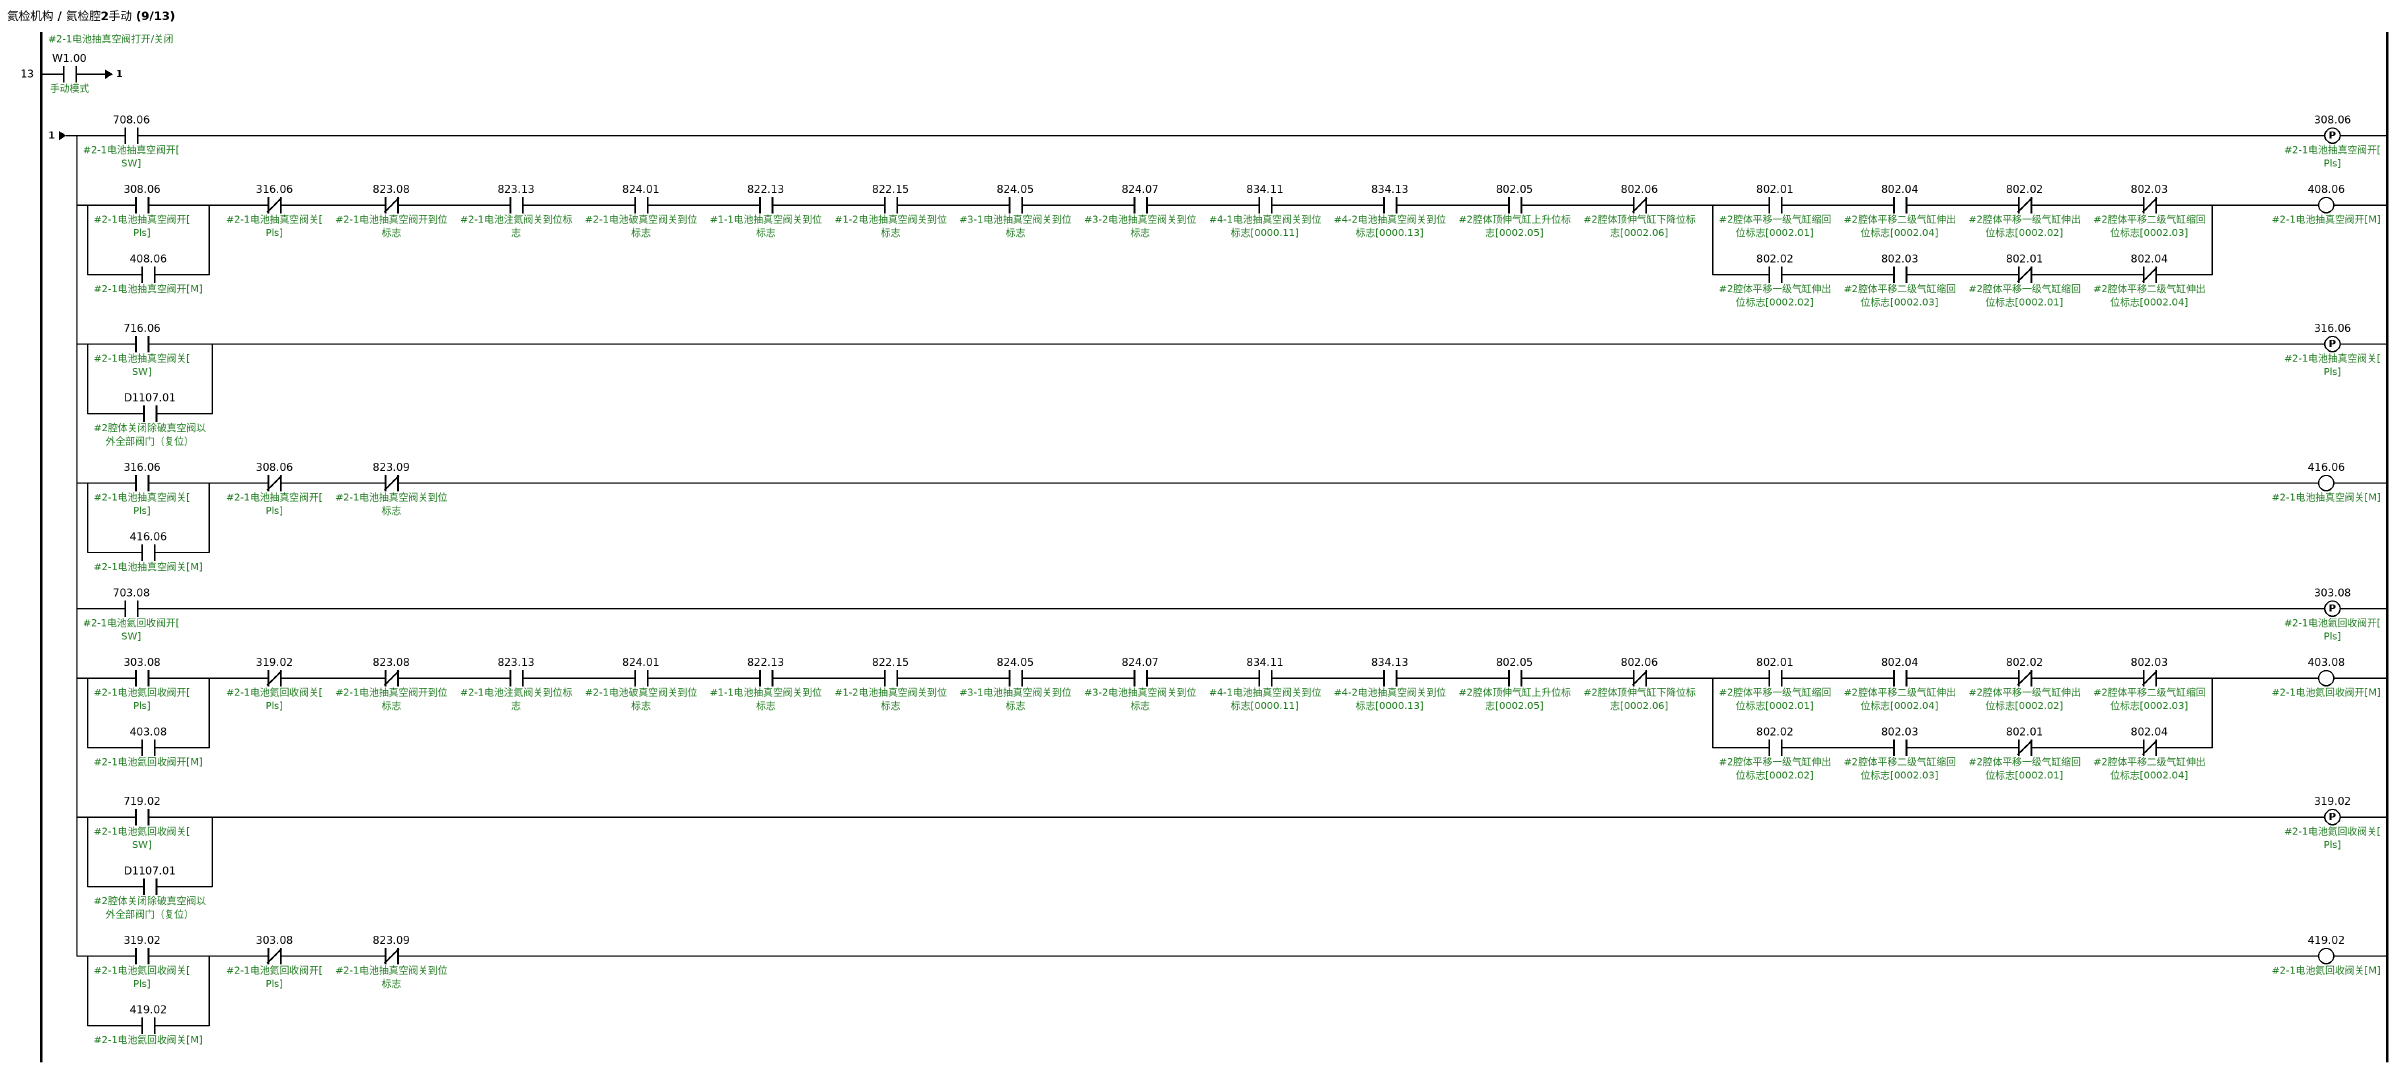
; [picture p192: 氦检机构 / 氦检腔2手动, rungs 13-13]
; rung 13: #2-1电池抽真空阀打开/关闭
LD W1.00  ; 手动模式
OUT TR0
AND 708.06  ; #2-1电池抽真空阀开[SW]
DIFU(013) 308.06  ; #2-1电池抽真空阀开[Pls]
LD TR0
LD 308.06  ; #2-1电池抽真空阀开[Pls]
OR 408.06  ; #2-1电池抽真空阀开[M]
ANDLD
ANDNOT 316.06  ; #2-1电池抽真空阀关[Pls]
ANDNOT 823.08  ; #2-1电池抽真空阀开到位标志
AND 823.13  ; #2-1电池注氦阀关到位标志
AND 824.01  ; #2-1电池破真空阀关到位标志
AND 822.13  ; #1-1电池抽真空阀关到位标志
AND 822.15  ; #1-2电池抽真空阀关到位标志
AND 824.05  ; #3-1电池抽真空阀关到位标志
AND 824.07  ; #3-2电池抽真空阀关到位标志
AND 834.11  ; #4-1电池抽真空阀关到位标志[0000.11]
AND 834.13  ; #4-2电池抽真空阀关到位标志[0000.13]
AND 802.05  ; #2腔体顶伸气缸上升位标志[0002.05]
ANDNOT 802.06  ; #2腔体顶伸气缸下降位标志[0002.06]
LD 802.01  ; #2腔体平移一级气缸缩回位标志[0002.01]
AND 802.04  ; #2腔体平移二级气缸伸出位标志[0002.04]
ANDNOT 802.02  ; #2腔体平移一级气缸伸出位标志[0002.02]
ANDNOT 802.03  ; #2腔体平移二级气缸缩回位标志[0002.03]
LD 802.02  ; #2腔体平移一级气缸伸出位标志[0002.02]
AND 802.03  ; #2腔体平移二级气缸缩回位标志[0002.03]
ANDNOT 802.01  ; #2腔体平移一级气缸缩回位标志[0002.01]
ANDNOT 802.04  ; #2腔体平移二级气缸伸出位标志[0002.04]
ORLD
ANDLD
OUT 408.06  ; #2-1电池抽真空阀开[M]
LD TR0
LD 716.06  ; #2-1电池抽真空阀关[SW]
OR D1107.01  ; #2腔体关闭除破真空阀以外全部阀门（复位）
ANDLD
DIFU(013) 316.06  ; #2-1电池抽真空阀关[Pls]
LD TR0
LD 316.06  ; #2-1电池抽真空阀关[Pls]
OR 416.06  ; #2-1电池抽真空阀关[M]
ANDLD
ANDNOT 308.06  ; #2-1电池抽真空阀开[Pls]
ANDNOT 823.09  ; #2-1电池抽真空阀关到位标志
OUT 416.06  ; #2-1电池抽真空阀关[M]
LD TR0
AND 703.08  ; #2-1电池氦回收阀开[SW]
DIFU(013) 303.08  ; #2-1电池氦回收阀开[Pls]
LD TR0
LD 303.08  ; #2-1电池氦回收阀开[Pls]
OR 403.08  ; #2-1电池氦回收阀开[M]
ANDLD
ANDNOT 319.02  ; #2-1电池氦回收阀关[Pls]
ANDNOT 823.08  ; #2-1电池抽真空阀开到位标志
AND 823.13  ; #2-1电池注氦阀关到位标志
AND 824.01  ; #2-1电池破真空阀关到位标志
AND 822.13  ; #1-1电池抽真空阀关到位标志
AND 822.15  ; #1-2电池抽真空阀关到位标志
AND 824.05  ; #3-1电池抽真空阀关到位标志
AND 824.07  ; #3-2电池抽真空阀关到位标志
AND 834.11  ; #4-1电池抽真空阀关到位标志[0000.11]
AND 834.13  ; #4-2电池抽真空阀关到位标志[0000.13]
AND 802.05  ; #2腔体顶伸气缸上升位标志[0002.05]
ANDNOT 802.06  ; #2腔体顶伸气缸下降位标志[0002.06]
LD 802.01  ; #2腔体平移一级气缸缩回位标志[0002.01]
AND 802.04  ; #2腔体平移二级气缸伸出位标志[0002.04]
ANDNOT 802.02  ; #2腔体平移一级气缸伸出位标志[0002.02]
ANDNOT 802.03  ; #2腔体平移二级气缸缩回位标志[0002.03]
LD 802.02  ; #2腔体平移一级气缸伸出位标志[0002.02]
AND 802.03  ; #2腔体平移二级气缸缩回位标志[0002.03]
ANDNOT 802.01  ; #2腔体平移一级气缸缩回位标志[0002.01]
ANDNOT 802.04  ; #2腔体平移二级气缸伸出位标志[0002.04]
ORLD
ANDLD
OUT 403.08  ; #2-1电池氦回收阀开[M]
LD TR0
LD 719.02  ; #2-1电池氦回收阀关[SW]
OR D1107.01  ; #2腔体关闭除破真空阀以外全部阀门（复位）
ANDLD
DIFU(013) 319.02  ; #2-1电池氦回收阀关[Pls]
LD TR0
LD 319.02  ; #2-1电池氦回收阀关[Pls]
OR 419.02  ; #2-1电池氦回收阀关[M]
ANDLD
ANDNOT 303.08  ; #2-1电池氦回收阀开[Pls]
ANDNOT 823.09  ; #2-1电池抽真空阀关到位标志
OUT 419.02  ; #2-1电池氦回收阀关[M]

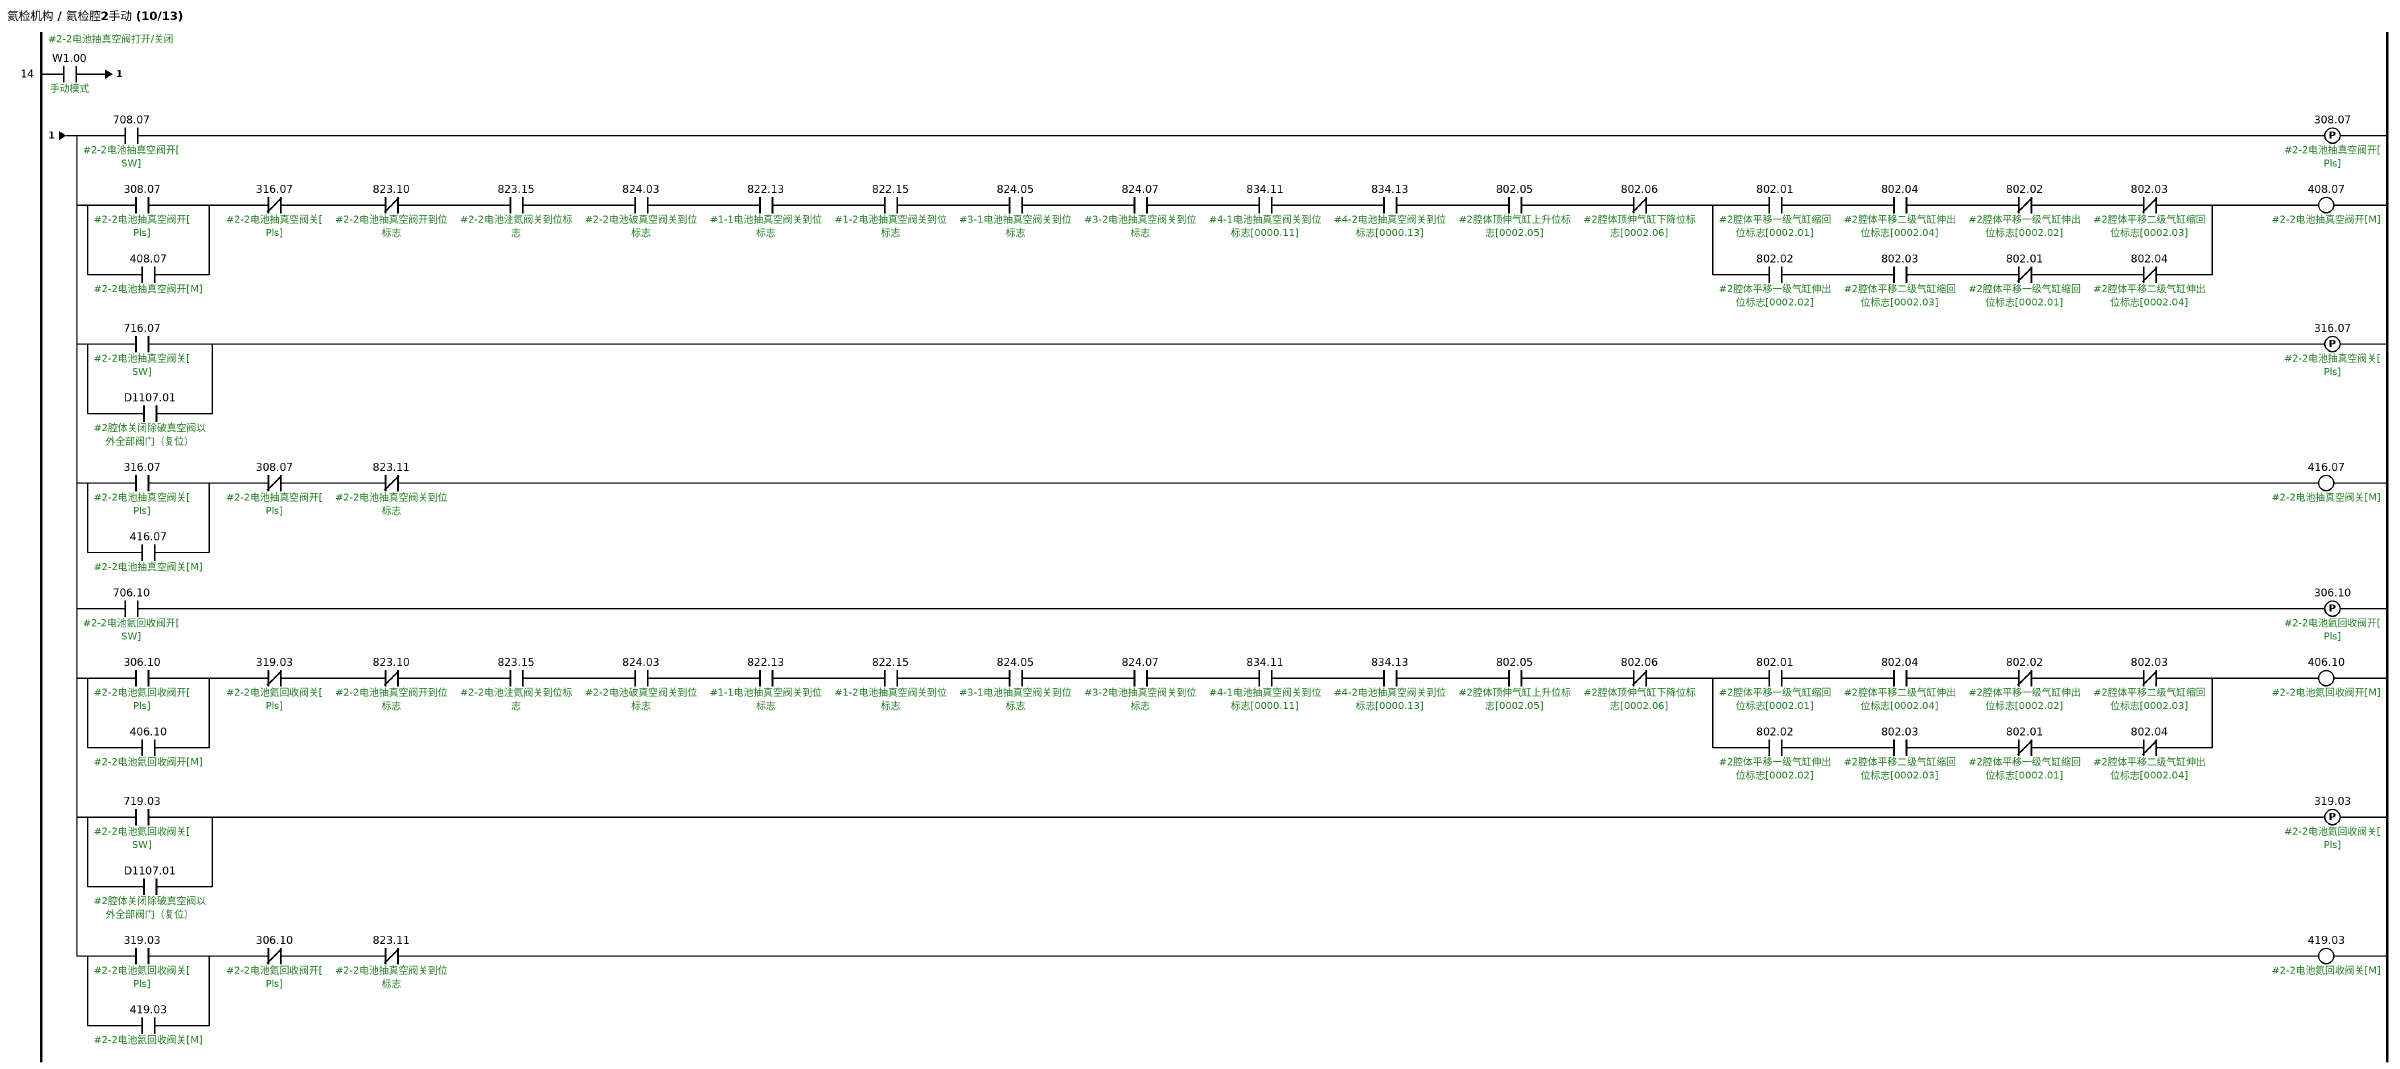
; rung 14: #2-2电池抽真空阀打开/关闭
LD W1.00  ; 手动模式
OUT TR0
AND 708.07  ; #2-2电池抽真空阀开[SW]
DIFU(013) 308.07  ; #2-2电池抽真空阀开[Pls]
LD TR0
LD 308.07  ; #2-2电池抽真空阀开[Pls]
OR 408.07  ; #2-2电池抽真空阀开[M]
ANDLD
ANDNOT 316.07  ; #2-2电池抽真空阀关[Pls]
ANDNOT 823.10  ; #2-2电池抽真空阀开到位标志
AND 823.15  ; #2-2电池注氦阀关到位标志
AND 824.03  ; #2-2电池破真空阀关到位标志
AND 822.13  ; #1-1电池抽真空阀关到位标志
AND 822.15  ; #1-2电池抽真空阀关到位标志
AND 824.05  ; #3-1电池抽真空阀关到位标志
AND 824.07  ; #3-2电池抽真空阀关到位标志
AND 834.11  ; #4-1电池抽真空阀关到位标志[0000.11]
AND 834.13  ; #4-2电池抽真空阀关到位标志[0000.13]
AND 802.05  ; #2腔体顶伸气缸上升位标志[0002.05]
ANDNOT 802.06  ; #2腔体顶伸气缸下降位标志[0002.06]
LD 802.01  ; #2腔体平移一级气缸缩回位标志[0002.01]
AND 802.04  ; #2腔体平移二级气缸伸出位标志[0002.04]
ANDNOT 802.02  ; #2腔体平移一级气缸伸出位标志[0002.02]
ANDNOT 802.03  ; #2腔体平移二级气缸缩回位标志[0002.03]
LD 802.02  ; #2腔体平移一级气缸伸出位标志[0002.02]
AND 802.03  ; #2腔体平移二级气缸缩回位标志[0002.03]
ANDNOT 802.01  ; #2腔体平移一级气缸缩回位标志[0002.01]
ANDNOT 802.04  ; #2腔体平移二级气缸伸出位标志[0002.04]
ORLD
ANDLD
OUT 408.07  ; #2-2电池抽真空阀开[M]
LD TR0
LD 716.07  ; #2-2电池抽真空阀关[SW]
OR D1107.01  ; #2腔体关闭除破真空阀以外全部阀门（复位）
ANDLD
DIFU(013) 316.07  ; #2-2电池抽真空阀关[Pls]
LD TR0
LD 316.07  ; #2-2电池抽真空阀关[Pls]
OR 416.07  ; #2-2电池抽真空阀关[M]
ANDLD
ANDNOT 308.07  ; #2-2电池抽真空阀开[Pls]
ANDNOT 823.11  ; #2-2电池抽真空阀关到位标志
OUT 416.07  ; #2-2电池抽真空阀关[M]
LD TR0
AND 706.10  ; #2-2电池氦回收阀开[SW]
DIFU(013) 306.10  ; #2-2电池氦回收阀开[Pls]
LD TR0
LD 306.10  ; #2-2电池氦回收阀开[Pls]
OR 406.10  ; #2-2电池氦回收阀开[M]
ANDLD
ANDNOT 319.03  ; #2-2电池氦回收阀关[Pls]
ANDNOT 823.10  ; #2-2电池抽真空阀开到位标志
AND 823.15  ; #2-2电池注氦阀关到位标志
AND 824.03  ; #2-2电池破真空阀关到位标志
AND 822.13  ; #1-1电池抽真空阀关到位标志
AND 822.15  ; #1-2电池抽真空阀关到位标志
AND 824.05  ; #3-1电池抽真空阀关到位标志
AND 824.07  ; #3-2电池抽真空阀关到位标志
AND 834.11  ; #4-1电池抽真空阀关到位标志[0000.11]
AND 834.13  ; #4-2电池抽真空阀关到位标志[0000.13]
AND 802.05  ; #2腔体顶伸气缸上升位标志[0002.05]
ANDNOT 802.06  ; #2腔体顶伸气缸下降位标志[0002.06]
LD 802.01  ; #2腔体平移一级气缸缩回位标志[0002.01]
AND 802.04  ; #2腔体平移二级气缸伸出位标志[0002.04]
ANDNOT 802.02  ; #2腔体平移一级气缸伸出位标志[0002.02]
ANDNOT 802.03  ; #2腔体平移二级气缸缩回位标志[0002.03]
LD 802.02  ; #2腔体平移一级气缸伸出位标志[0002.02]
AND 802.03  ; #2腔体平移二级气缸缩回位标志[0002.03]
ANDNOT 802.01  ; #2腔体平移一级气缸缩回位标志[0002.01]
ANDNOT 802.04  ; #2腔体平移二级气缸伸出位标志[0002.04]
ORLD
ANDLD
OUT 406.10  ; #2-2电池氦回收阀开[M]
LD TR0
LD 719.03  ; #2-2电池氦回收阀关[SW]
OR D1107.01  ; #2腔体关闭除破真空阀以外全部阀门（复位）
ANDLD
DIFU(013) 319.03  ; #2-2电池氦回收阀关[Pls]
LD TR0
LD 319.03  ; #2-2电池氦回收阀关[Pls]
OR 419.03  ; #2-2电池氦回收阀关[M]
ANDLD
ANDNOT 306.10  ; #2-2电池氦回收阀开[Pls]
ANDNOT 823.11  ; #2-2电池抽真空阀关到位标志
OUT 419.03  ; #2-2电池氦回收阀关[M]

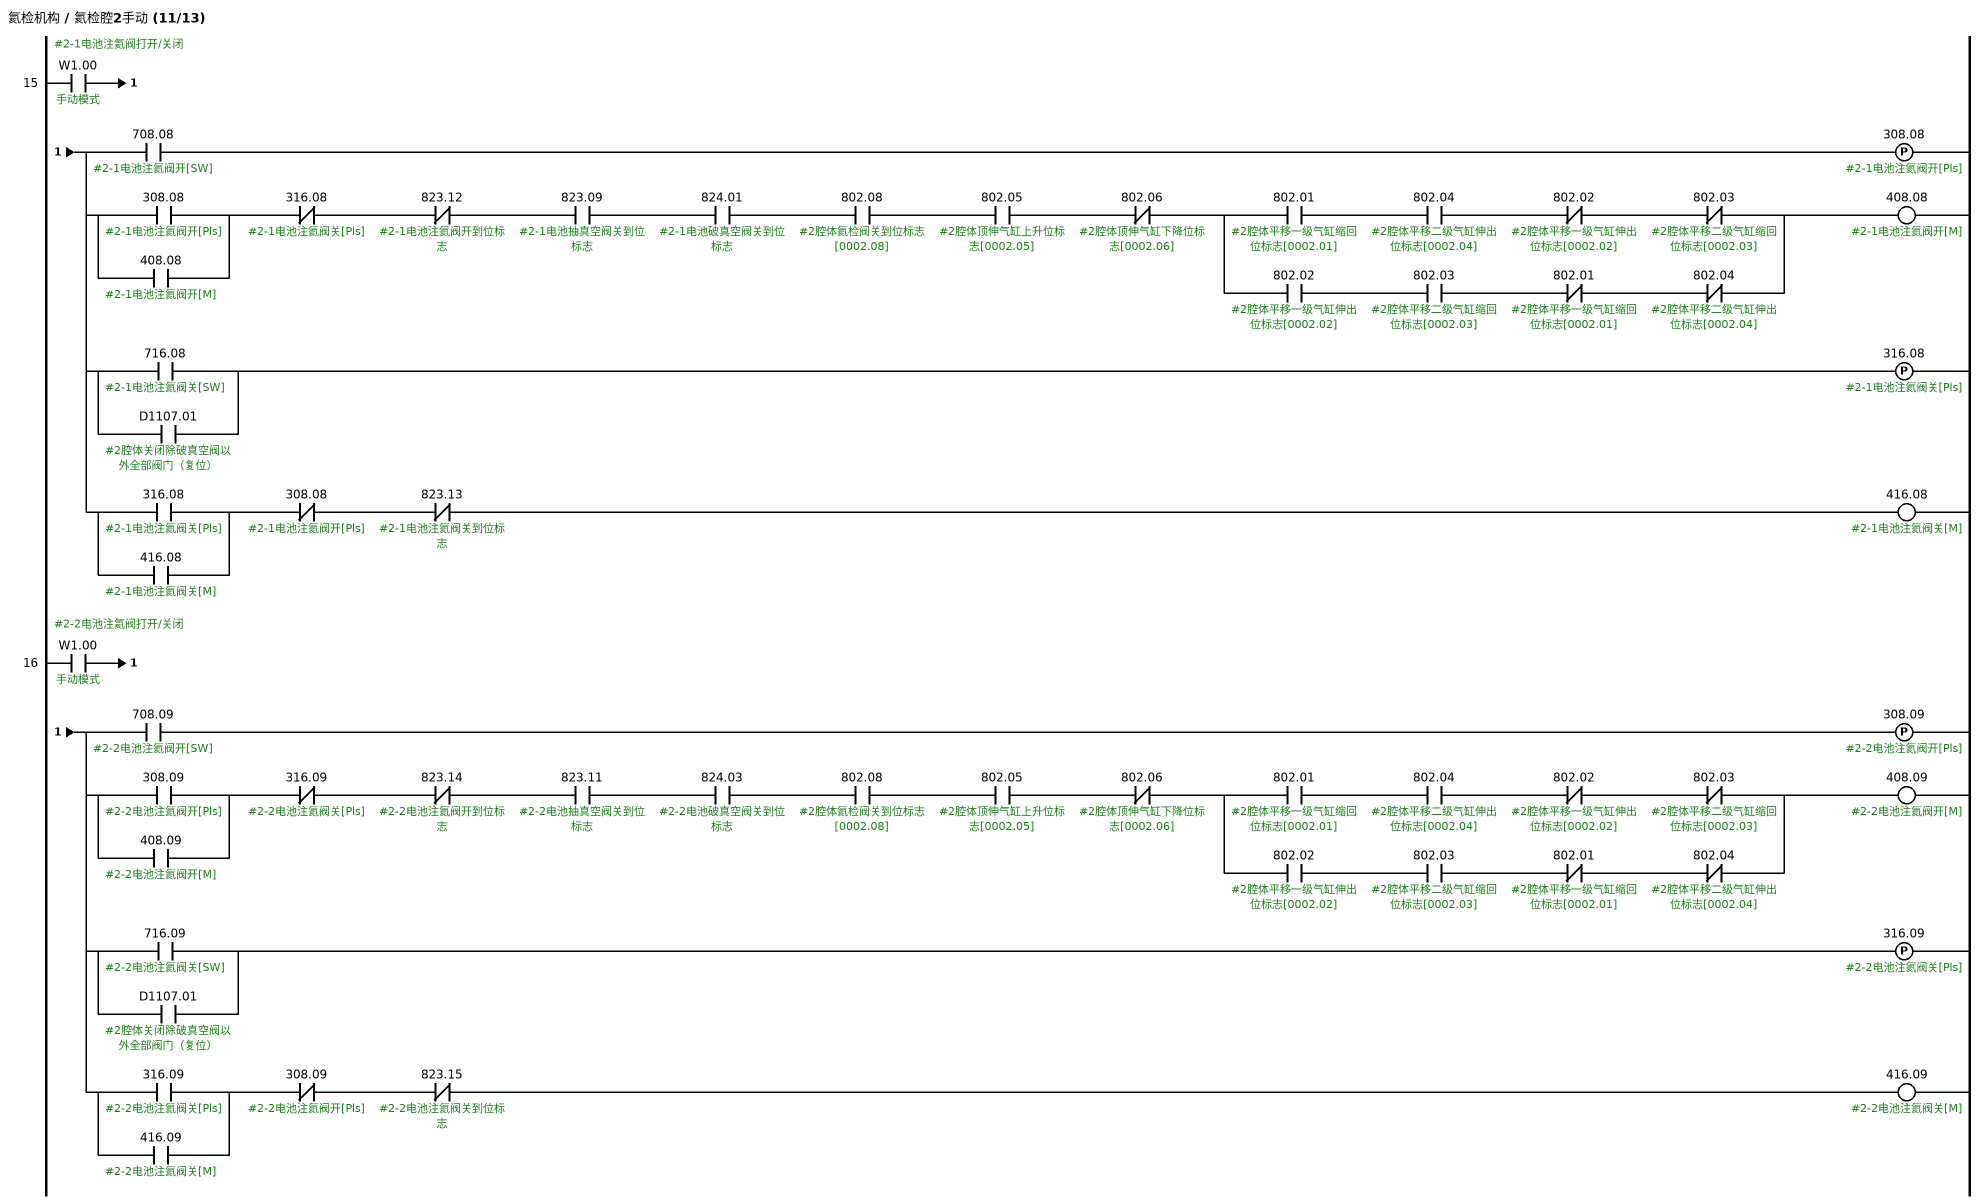
; rung 15: #2-1电池注氦阀打开/关闭
LD W1.00  ; 手动模式
OUT TR0
AND 708.08  ; #2-1电池注氦阀开[SW]
DIFU(013) 308.08  ; #2-1电池注氦阀开[Pls]
LD TR0
LD 308.08  ; #2-1电池注氦阀开[Pls]
OR 408.08  ; #2-1电池注氦阀开[M]
ANDLD
ANDNOT 316.08  ; #2-1电池注氦阀关[Pls]
ANDNOT 823.12  ; #2-1电池注氦阀开到位标志
AND 823.09  ; #2-1电池抽真空阀关到位标志
AND 824.01  ; #2-1电池破真空阀关到位标志
AND 802.08  ; #2腔体氦检阀关到位标志[0002.08]
AND 802.05  ; #2腔体顶伸气缸上升位标志[0002.05]
ANDNOT 802.06  ; #2腔体顶伸气缸下降位标志[0002.06]
LD 802.01  ; #2腔体平移一级气缸缩回位标志[0002.01]
AND 802.04  ; #2腔体平移二级气缸伸出位标志[0002.04]
ANDNOT 802.02  ; #2腔体平移一级气缸伸出位标志[0002.02]
ANDNOT 802.03  ; #2腔体平移二级气缸缩回位标志[0002.03]
LD 802.02  ; #2腔体平移一级气缸伸出位标志[0002.02]
AND 802.03  ; #2腔体平移二级气缸缩回位标志[0002.03]
ANDNOT 802.01  ; #2腔体平移一级气缸缩回位标志[0002.01]
ANDNOT 802.04  ; #2腔体平移二级气缸伸出位标志[0002.04]
ORLD
ANDLD
OUT 408.08  ; #2-1电池注氦阀开[M]
LD TR0
LD 716.08  ; #2-1电池注氦阀关[SW]
OR D1107.01  ; #2腔体关闭除破真空阀以外全部阀门（复位）
ANDLD
DIFU(013) 316.08  ; #2-1电池注氦阀关[Pls]
LD TR0
LD 316.08  ; #2-1电池注氦阀关[Pls]
OR 416.08  ; #2-1电池注氦阀关[M]
ANDLD
ANDNOT 308.08  ; #2-1电池注氦阀开[Pls]
ANDNOT 823.13  ; #2-1电池注氦阀关到位标志
OUT 416.08  ; #2-1电池注氦阀关[M]
; rung 16: #2-2电池注氦阀打开/关闭
LD W1.00  ; 手动模式
OUT TR0
AND 708.09  ; #2-2电池注氦阀开[SW]
DIFU(013) 308.09  ; #2-2电池注氦阀开[Pls]
LD TR0
LD 308.09  ; #2-2电池注氦阀开[Pls]
OR 408.09  ; #2-2电池注氦阀开[M]
ANDLD
ANDNOT 316.09  ; #2-2电池注氦阀关[Pls]
ANDNOT 823.14  ; #2-2电池注氦阀开到位标志
AND 823.11  ; #2-2电池抽真空阀关到位标志
AND 824.03  ; #2-2电池破真空阀关到位标志
AND 802.08  ; #2腔体氦检阀关到位标志[0002.08]
AND 802.05  ; #2腔体顶伸气缸上升位标志[0002.05]
ANDNOT 802.06  ; #2腔体顶伸气缸下降位标志[0002.06]
LD 802.01  ; #2腔体平移一级气缸缩回位标志[0002.01]
AND 802.04  ; #2腔体平移二级气缸伸出位标志[0002.04]
ANDNOT 802.02  ; #2腔体平移一级气缸伸出位标志[0002.02]
ANDNOT 802.03  ; #2腔体平移二级气缸缩回位标志[0002.03]
LD 802.02  ; #2腔体平移一级气缸伸出位标志[0002.02]
AND 802.03  ; #2腔体平移二级气缸缩回位标志[0002.03]
ANDNOT 802.01  ; #2腔体平移一级气缸缩回位标志[0002.01]
ANDNOT 802.04  ; #2腔体平移二级气缸伸出位标志[0002.04]
ORLD
ANDLD
OUT 408.09  ; #2-2电池注氦阀开[M]
LD TR0
LD 716.09  ; #2-2电池注氦阀关[SW]
OR D1107.01  ; #2腔体关闭除破真空阀以外全部阀门（复位）
ANDLD
DIFU(013) 316.09  ; #2-2电池注氦阀关[Pls]
LD TR0
LD 316.09  ; #2-2电池注氦阀关[Pls]
OR 416.09  ; #2-2电池注氦阀关[M]
ANDLD
ANDNOT 308.09  ; #2-2电池注氦阀开[Pls]
ANDNOT 823.15  ; #2-2电池注氦阀关到位标志
OUT 416.09  ; #2-2电池注氦阀关[M]

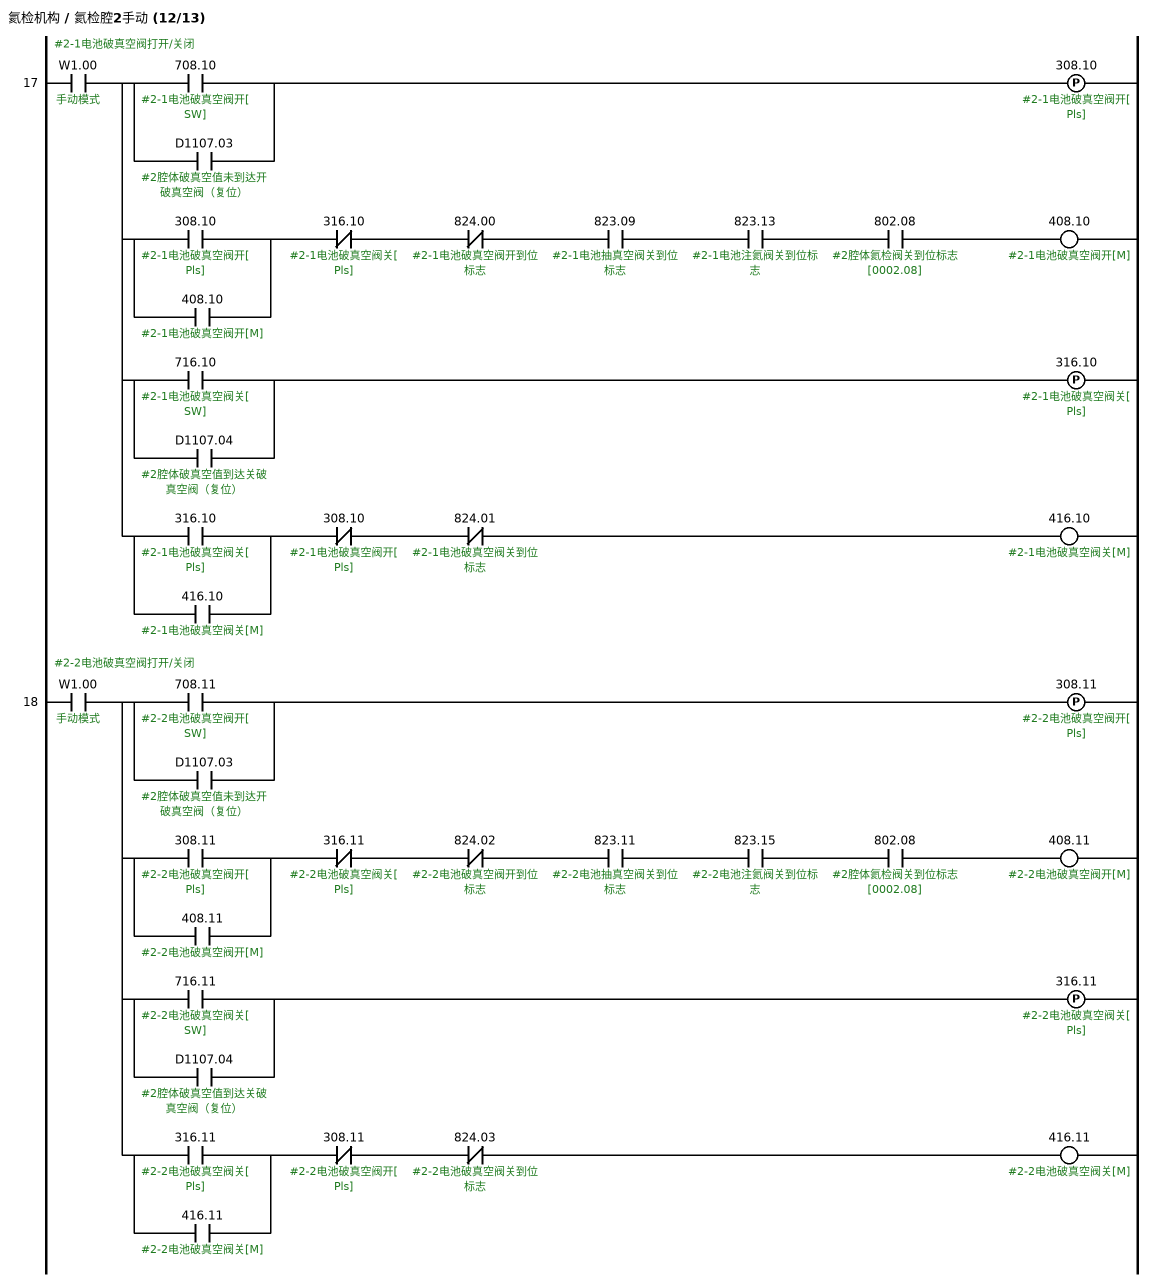
; rung 17: #2-1电池破真空阀打开/关闭
LD W1.00  ; 手动模式
OUT TR0
LD 708.10  ; #2-1电池破真空阀开[SW]
OR D1107.03  ; #2腔体破真空值未到达开破真空阀（复位）
ANDLD
DIFU(013) 308.10  ; #2-1电池破真空阀开[Pls]
LD TR0
LD 308.10  ; #2-1电池破真空阀开[Pls]
OR 408.10  ; #2-1电池破真空阀开[M]
ANDLD
ANDNOT 316.10  ; #2-1电池破真空阀关[Pls]
ANDNOT 824.00  ; #2-1电池破真空阀开到位标志
AND 823.09  ; #2-1电池抽真空阀关到位标志
AND 823.13  ; #2-1电池注氦阀关到位标志
AND 802.08  ; #2腔体氦检阀关到位标志[0002.08]
OUT 408.10  ; #2-1电池破真空阀开[M]
LD TR0
LD 716.10  ; #2-1电池破真空阀关[SW]
OR D1107.04  ; #2腔体破真空值到达关破真空阀（复位）
ANDLD
DIFU(013) 316.10  ; #2-1电池破真空阀关[Pls]
LD TR0
LD 316.10  ; #2-1电池破真空阀关[Pls]
OR 416.10  ; #2-1电池破真空阀关[M]
ANDLD
ANDNOT 308.10  ; #2-1电池破真空阀开[Pls]
ANDNOT 824.01  ; #2-1电池破真空阀关到位标志
OUT 416.10  ; #2-1电池破真空阀关[M]
; rung 18: #2-2电池破真空阀打开/关闭
LD W1.00  ; 手动模式
OUT TR0
LD 708.11  ; #2-2电池破真空阀开[SW]
OR D1107.03  ; #2腔体破真空值未到达开破真空阀（复位）
ANDLD
DIFU(013) 308.11  ; #2-2电池破真空阀开[Pls]
LD TR0
LD 308.11  ; #2-2电池破真空阀开[Pls]
OR 408.11  ; #2-2电池破真空阀开[M]
ANDLD
ANDNOT 316.11  ; #2-2电池破真空阀关[Pls]
ANDNOT 824.02  ; #2-2电池破真空阀开到位标志
AND 823.11  ; #2-2电池抽真空阀关到位标志
AND 823.15  ; #2-2电池注氦阀关到位标志
AND 802.08  ; #2腔体氦检阀关到位标志[0002.08]
OUT 408.11  ; #2-2电池破真空阀开[M]
LD TR0
LD 716.11  ; #2-2电池破真空阀关[SW]
OR D1107.04  ; #2腔体破真空值到达关破真空阀（复位）
ANDLD
DIFU(013) 316.11  ; #2-2电池破真空阀关[Pls]
LD TR0
LD 316.11  ; #2-2电池破真空阀关[Pls]
OR 416.11  ; #2-2电池破真空阀关[M]
ANDLD
ANDNOT 308.11  ; #2-2电池破真空阀开[Pls]
ANDNOT 824.03  ; #2-2电池破真空阀关到位标志
OUT 416.11  ; #2-2电池破真空阀关[M]

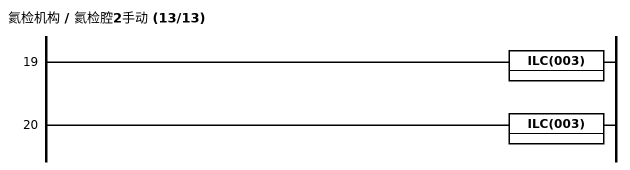
; rung 19
ILC(003)
; rung 20
ILC(003)

### Section 氦检腔3手动

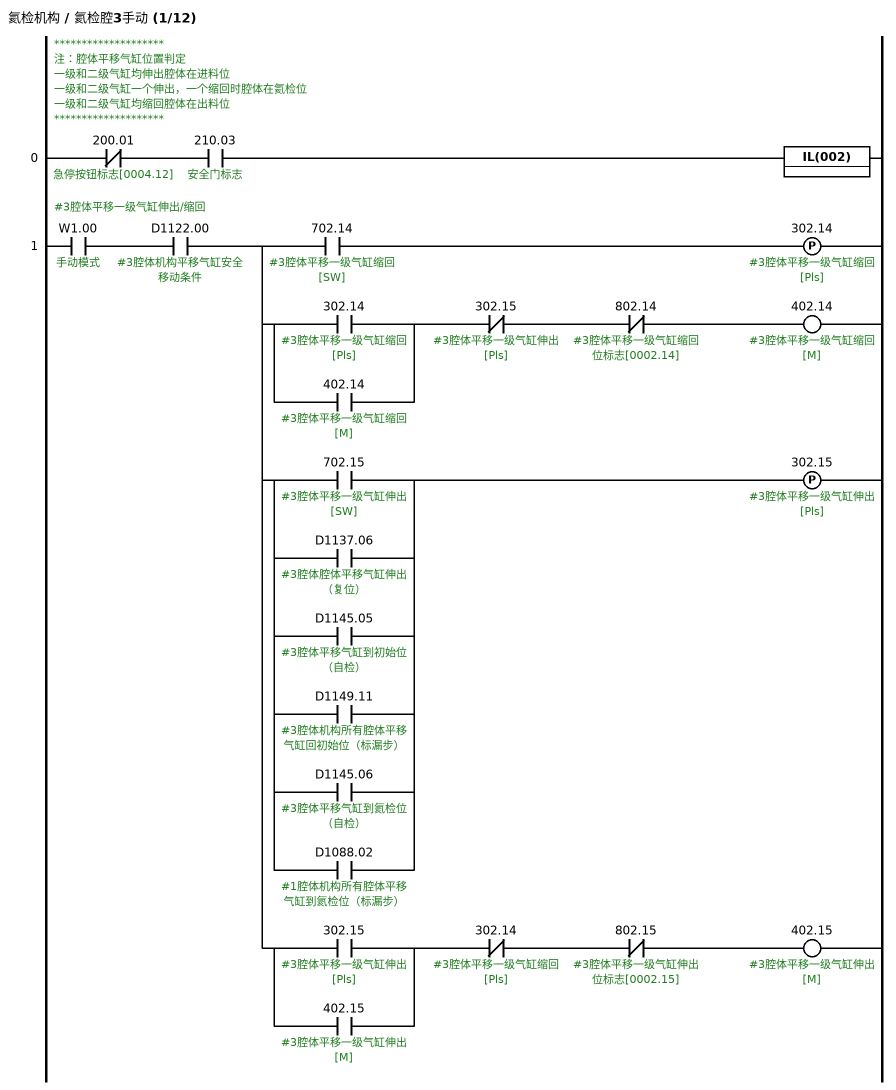
; rung 0: ******************** / 注：腔体平移气缸位置判定 / 一级和二级气缸均伸出腔体在进料位 / 一级和二级气缸一个伸出，一个缩回时腔体在氦检位 / 一级和二级气缸均缩回腔体在出料位 / ********************
LDNOT 200.01  ; 急停按钮标志[0004.12]
AND 210.03  ; 安全门标志
IL(002)
; rung 1: #3腔体平移一级气缸伸出/缩回
LD W1.00  ; 手动模式
AND D1122.00  ; #3腔体机构平移气缸安全移动条件
OUT TR0
AND 702.14  ; #3腔体平移一级气缸缩回[SW]
DIFU(013) 302.14  ; #3腔体平移一级气缸缩回[Pls]
LD TR0
LD 302.14  ; #3腔体平移一级气缸缩回[Pls]
OR 402.14  ; #3腔体平移一级气缸缩回[M]
ANDLD
ANDNOT 302.15  ; #3腔体平移一级气缸伸出[Pls]
ANDNOT 802.14  ; #3腔体平移一级气缸缩回位标志[0002.14]
OUT 402.14  ; #3腔体平移一级气缸缩回[M]
LD TR0
LD 702.15  ; #3腔体平移一级气缸伸出[SW]
OR D1137.06  ; #3腔体腔体平移气缸伸出（复位）
OR D1145.05  ; #3腔体平移气缸到初始位（自检）
OR D1149.11  ; #3腔体机构所有腔体平移气缸回初始位（标漏步）
OR D1145.06  ; #3腔体平移气缸到氦检位（自检）
OR D1088.02  ; #1腔体机构所有腔体平移气缸到氦检位（标漏步）
ANDLD
DIFU(013) 302.15  ; #3腔体平移一级气缸伸出[Pls]
LD TR0
LD 302.15  ; #3腔体平移一级气缸伸出[Pls]
OR 402.15  ; #3腔体平移一级气缸伸出[M]
ANDLD
ANDNOT 302.14  ; #3腔体平移一级气缸缩回[Pls]
ANDNOT 802.15  ; #3腔体平移一级气缸伸出位标志[0002.15]
OUT 402.15  ; #3腔体平移一级气缸伸出[M]

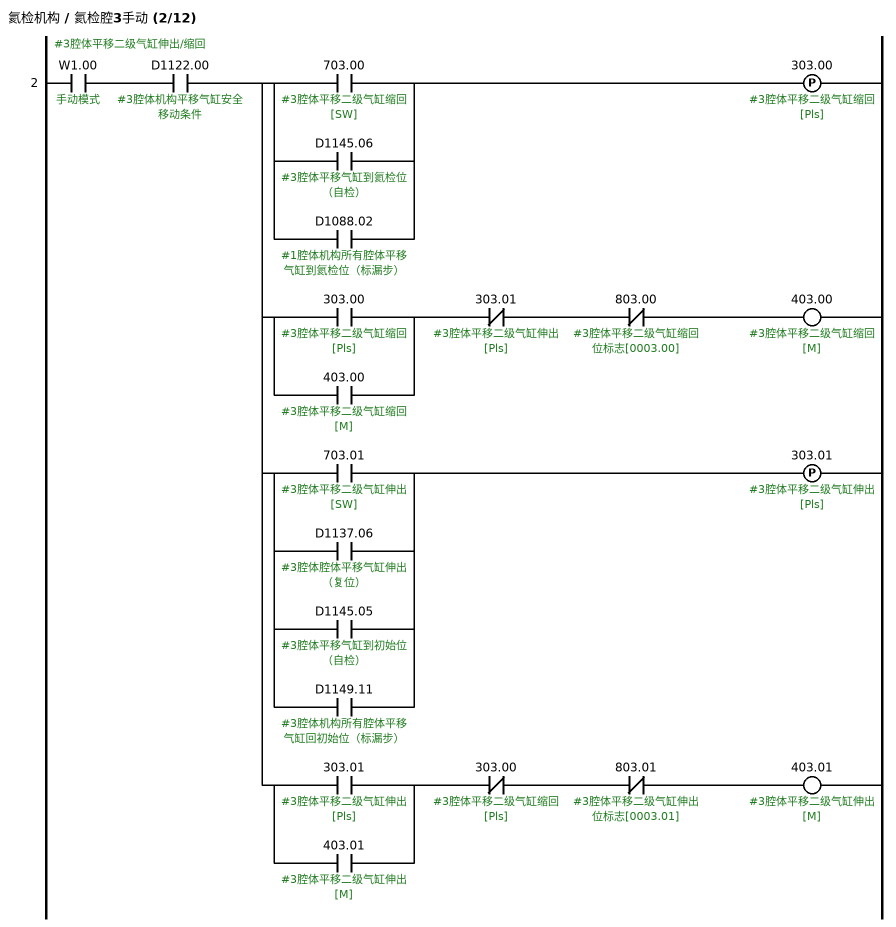
; rung 2: #3腔体平移二级气缸伸出/缩回
LD W1.00  ; 手动模式
AND D1122.00  ; #3腔体机构平移气缸安全移动条件
OUT TR0
LD 703.00  ; #3腔体平移二级气缸缩回[SW]
OR D1145.06  ; #3腔体平移气缸到氦检位（自检）
OR D1088.02  ; #1腔体机构所有腔体平移气缸到氦检位（标漏步）
ANDLD
DIFU(013) 303.00  ; #3腔体平移二级气缸缩回[Pls]
LD TR0
LD 303.00  ; #3腔体平移二级气缸缩回[Pls]
OR 403.00  ; #3腔体平移二级气缸缩回[M]
ANDLD
ANDNOT 303.01  ; #3腔体平移二级气缸伸出[Pls]
ANDNOT 803.00  ; #3腔体平移二级气缸缩回位标志[0003.00]
OUT 403.00  ; #3腔体平移二级气缸缩回[M]
LD TR0
LD 703.01  ; #3腔体平移二级气缸伸出[SW]
OR D1137.06  ; #3腔体腔体平移气缸伸出（复位）
OR D1145.05  ; #3腔体平移气缸到初始位（自检）
OR D1149.11  ; #3腔体机构所有腔体平移气缸回初始位（标漏步）
ANDLD
DIFU(013) 303.01  ; #3腔体平移二级气缸伸出[Pls]
LD TR0
LD 303.01  ; #3腔体平移二级气缸伸出[Pls]
OR 403.01  ; #3腔体平移二级气缸伸出[M]
ANDLD
ANDNOT 303.00  ; #3腔体平移二级气缸缩回[Pls]
ANDNOT 803.01  ; #3腔体平移二级气缸伸出位标志[0003.01]
OUT 403.01  ; #3腔体平移二级气缸伸出[M]

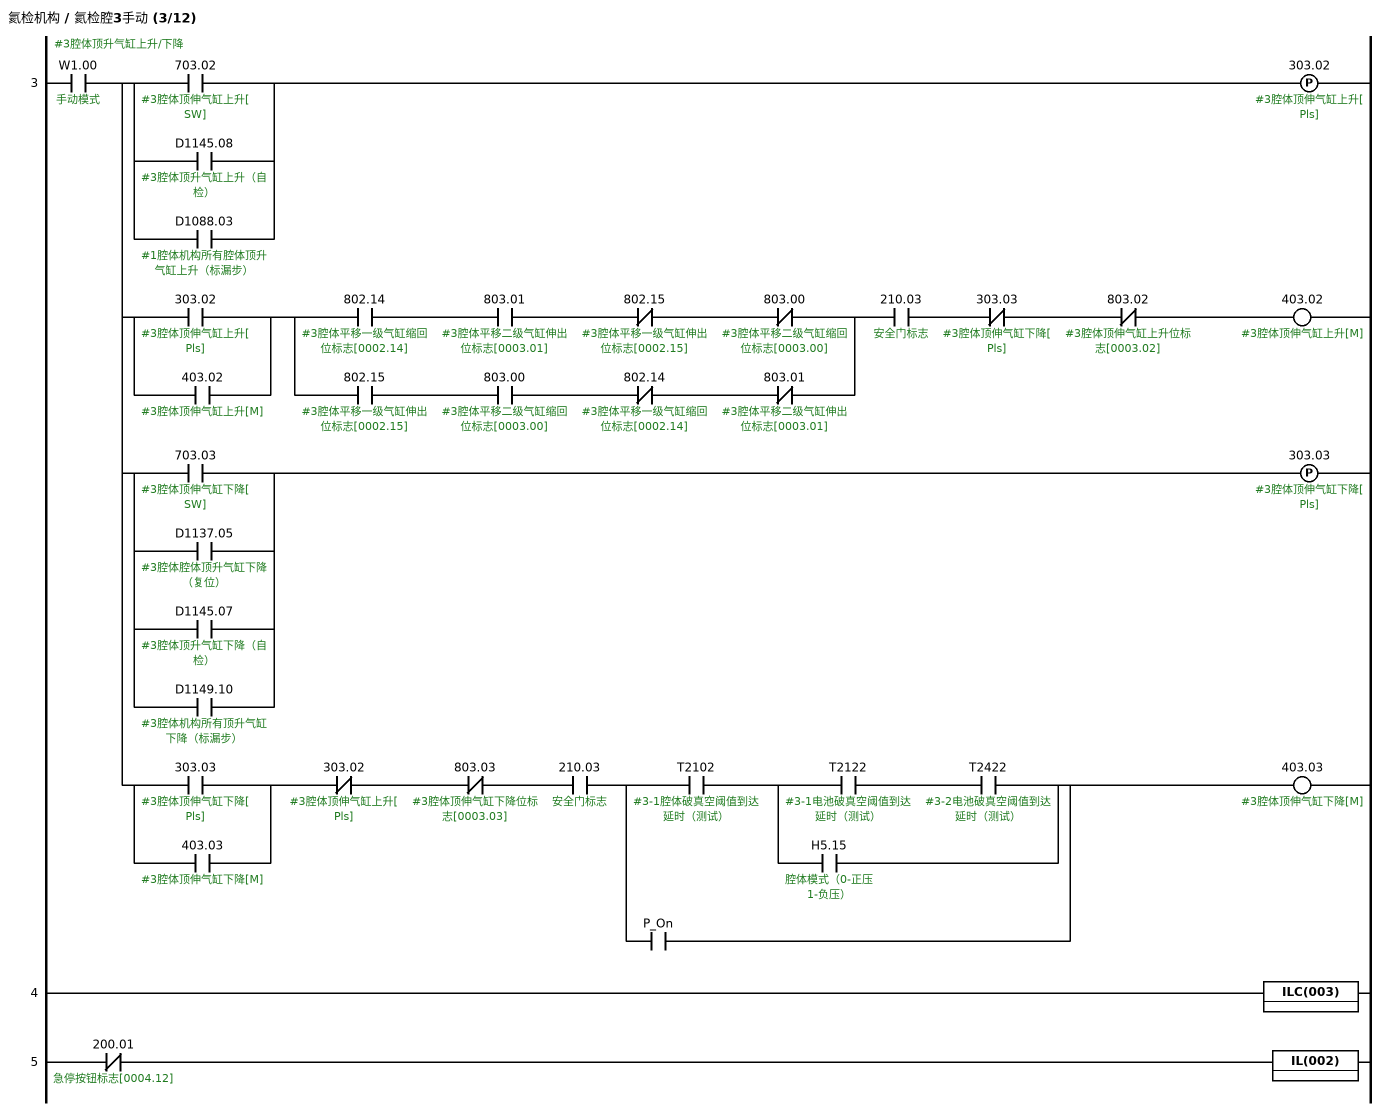
; rung 3: #3腔体顶升气缸上升/下降
LD W1.00  ; 手动模式
OUT TR0
LD 703.02  ; #3腔体顶伸气缸上升[SW]
OR D1145.08  ; #3腔体顶升气缸上升（自检）
OR D1088.03  ; #1腔体机构所有腔体顶升气缸上升（标漏步）
ANDLD
DIFU(013) 303.02  ; #3腔体顶伸气缸上升[Pls]
LD TR0
LD 303.02  ; #3腔体顶伸气缸上升[Pls]
OR 403.02  ; #3腔体顶伸气缸上升[M]
ANDLD
LD 802.14  ; #3腔体平移一级气缸缩回位标志[0002.14]
AND 803.01  ; #3腔体平移二级气缸伸出位标志[0003.01]
ANDNOT 802.15  ; #3腔体平移一级气缸伸出位标志[0002.15]
ANDNOT 803.00  ; #3腔体平移二级气缸缩回位标志[0003.00]
LD 802.15  ; #3腔体平移一级气缸伸出位标志[0002.15]
AND 803.00  ; #3腔体平移二级气缸缩回位标志[0003.00]
ANDNOT 802.14  ; #3腔体平移一级气缸缩回位标志[0002.14]
ANDNOT 803.01  ; #3腔体平移二级气缸伸出位标志[0003.01]
ORLD
ANDLD
AND 210.03  ; 安全门标志
ANDNOT 303.03  ; #3腔体顶伸气缸下降[Pls]
ANDNOT 803.02  ; #3腔体顶伸气缸上升位标志[0003.02]
OUT 403.02  ; #3腔体顶伸气缸上升[M]
LD TR0
LD 703.03  ; #3腔体顶伸气缸下降[SW]
OR D1137.05  ; #3腔体腔体顶升气缸下降（复位）
OR D1145.07  ; #3腔体顶升气缸下降（自检）
OR D1149.10  ; #3腔体机构所有顶升气缸下降（标漏步）
ANDLD
DIFU(013) 303.03  ; #3腔体顶伸气缸下降[Pls]
LD TR0
LD 303.03  ; #3腔体顶伸气缸下降[Pls]
OR 403.03  ; #3腔体顶伸气缸下降[M]
ANDLD
ANDNOT 303.02  ; #3腔体顶伸气缸上升[Pls]
ANDNOT 803.03  ; #3腔体顶伸气缸下降位标志[0003.03]
AND 210.03  ; 安全门标志
LD T2102  ; #3-1腔体破真空阈值到达延时（测试）
LD T2122  ; #3-1电池破真空阈值到达延时（测试）
AND T2422  ; #3-2电池破真空阈值到达延时（测试）
OR H5.15  ; 腔体模式（0-正压 1-负压）
ANDLD
OR P_On
ANDLD
OUT 403.03  ; #3腔体顶伸气缸下降[M]
; rung 4
ILC(003)
; rung 5
LDNOT 200.01  ; 急停按钮标志[0004.12]
IL(002)

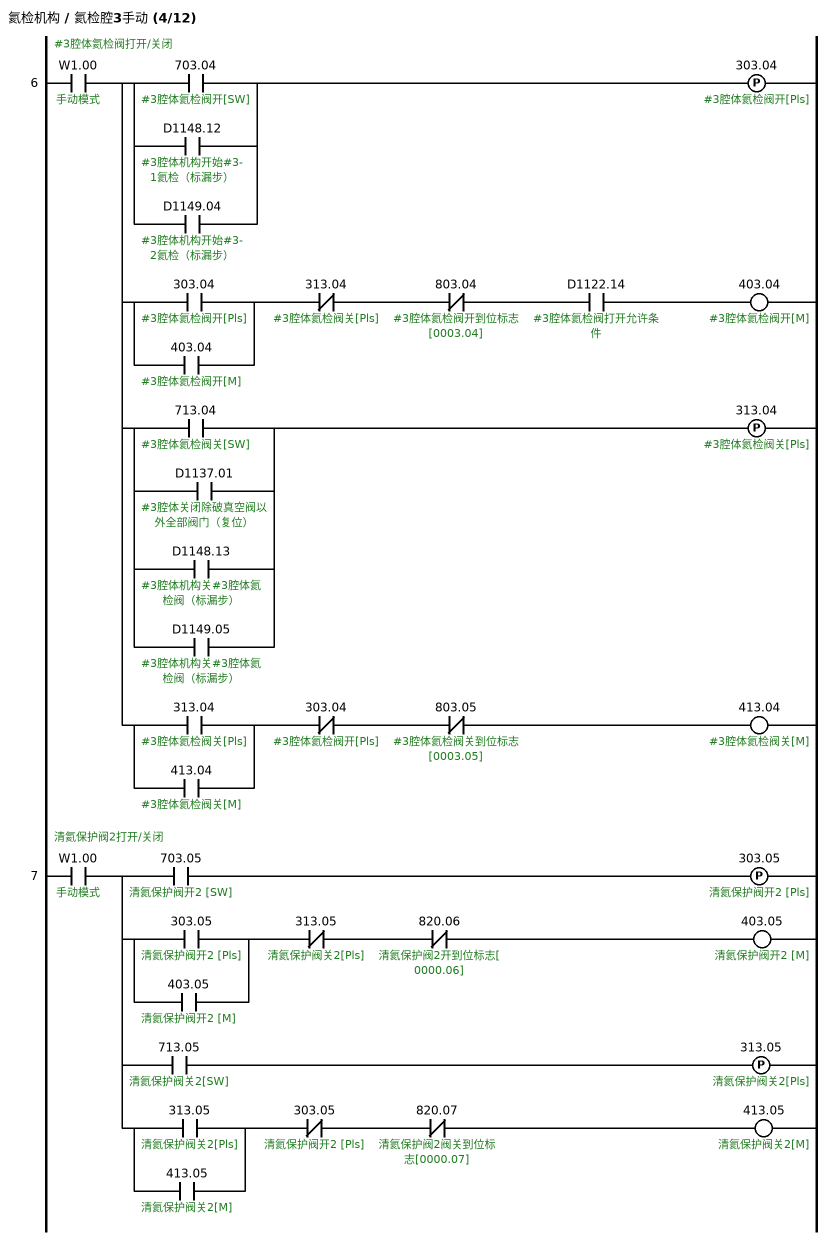
; rung 6: #3腔体氦检阀打开/关闭
LD W1.00  ; 手动模式
OUT TR0
LD 703.04  ; #3腔体氦检阀开[SW]
OR D1148.12  ; #3腔体机构开始#3-1氦检（标漏步）
OR D1149.04  ; #3腔体机构开始#3-2氦检（标漏步）
ANDLD
DIFU(013) 303.04  ; #3腔体氦检阀开[Pls]
LD TR0
LD 303.04  ; #3腔体氦检阀开[Pls]
OR 403.04  ; #3腔体氦检阀开[M]
ANDLD
ANDNOT 313.04  ; #3腔体氦检阀关[Pls]
ANDNOT 803.04  ; #3腔体氦检阀开到位标志[0003.04]
AND D1122.14  ; #3腔体氦检阀打开允许条件
OUT 403.04  ; #3腔体氦检阀开[M]
LD TR0
LD 713.04  ; #3腔体氦检阀关[SW]
OR D1137.01  ; #3腔体关闭除破真空阀以外全部阀门（复位）
OR D1148.13  ; #3腔体机构关#3腔体氦检阀（标漏步）
OR D1149.05  ; #3腔体机构关#3腔体氦检阀（标漏步）
ANDLD
DIFU(013) 313.04  ; #3腔体氦检阀关[Pls]
LD TR0
LD 313.04  ; #3腔体氦检阀关[Pls]
OR 413.04  ; #3腔体氦检阀关[M]
ANDLD
ANDNOT 303.04  ; #3腔体氦检阀开[Pls]
ANDNOT 803.05  ; #3腔体氦检阀关到位标志[0003.05]
OUT 413.04  ; #3腔体氦检阀关[M]
; rung 7: 清氦保护阀2打开/关闭
LD W1.00  ; 手动模式
OUT TR0
AND 703.05  ; 清氦保护阀开2 [SW]
DIFU(013) 303.05  ; 清氦保护阀开2 [Pls]
LD TR0
LD 303.05  ; 清氦保护阀开2 [Pls]
OR 403.05  ; 清氦保护阀开2 [M]
ANDLD
ANDNOT 313.05  ; 清氦保护阀关2[Pls]
ANDNOT 820.06  ; 清氦保护阀2开到位标志[0000.06]
OUT 403.05  ; 清氦保护阀开2 [M]
LD TR0
AND 713.05  ; 清氦保护阀关2[SW]
DIFU(013) 313.05  ; 清氦保护阀关2[Pls]
LD TR0
LD 313.05  ; 清氦保护阀关2[Pls]
OR 413.05  ; 清氦保护阀关2[M]
ANDLD
ANDNOT 303.05  ; 清氦保护阀开2 [Pls]
ANDNOT 820.07  ; 清氦保护阀2阀关到位标志[0000.07]
OUT 413.05  ; 清氦保护阀关2[M]

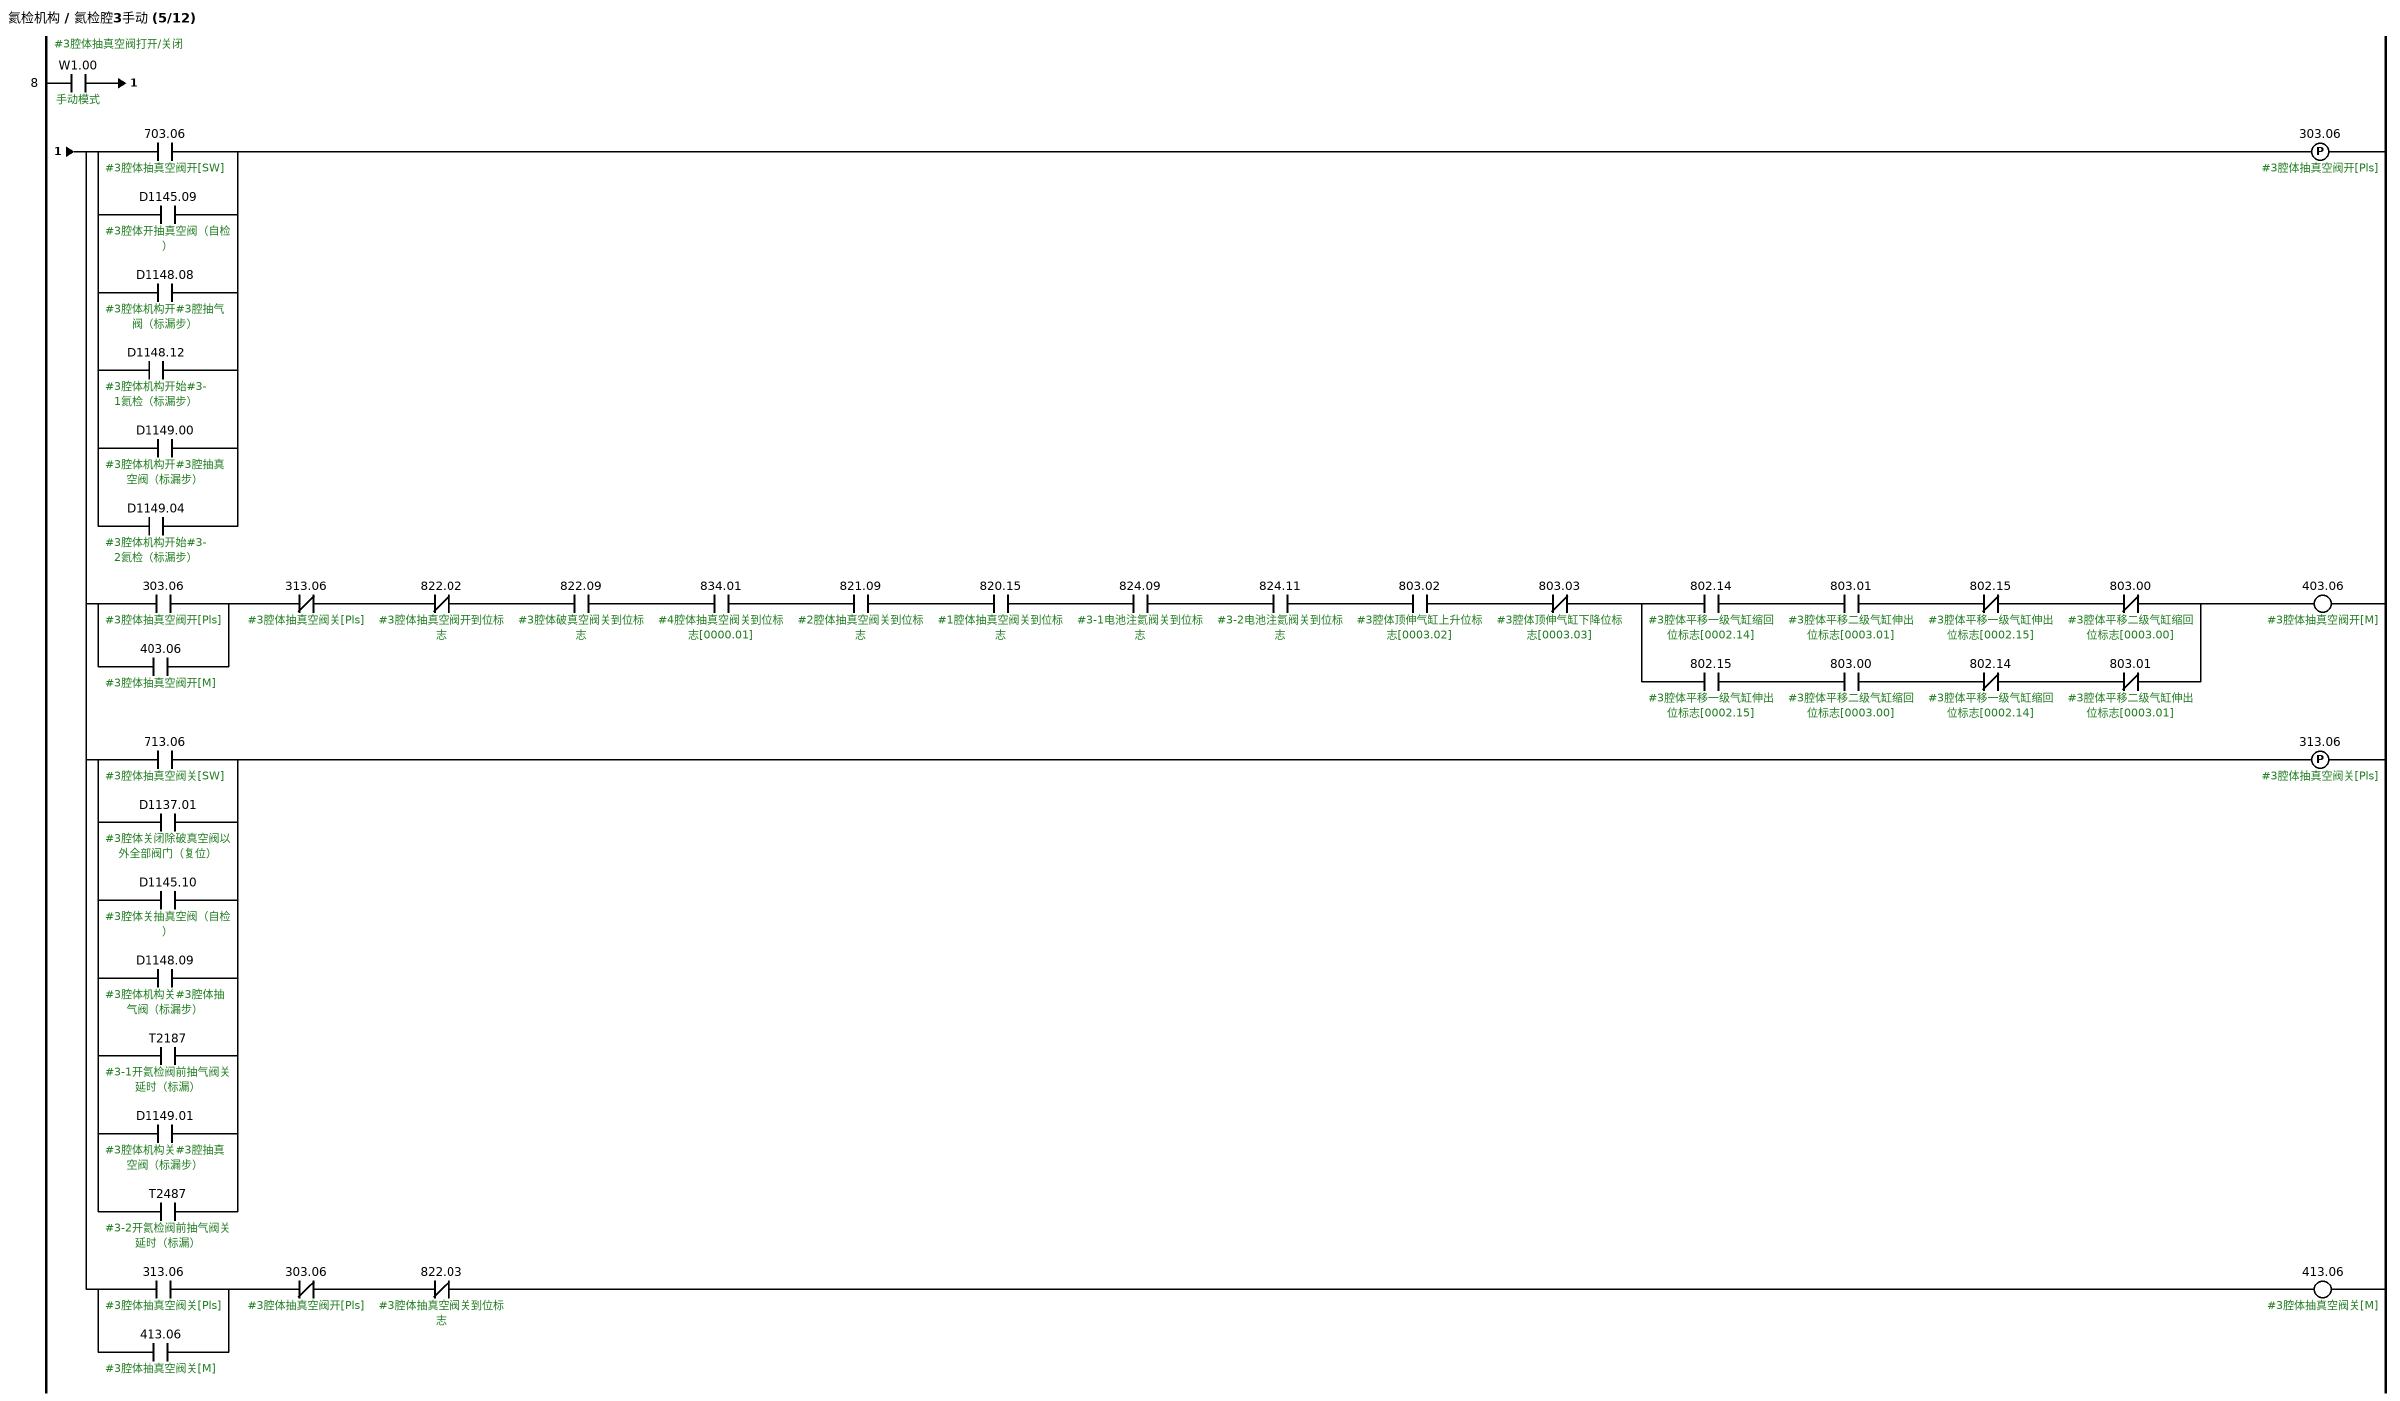
; rung 8: #3腔体抽真空阀打开/关闭
LD W1.00  ; 手动模式
OUT TR0
LD 703.06  ; #3腔体抽真空阀开[SW]
OR D1145.09  ; #3腔体开抽真空阀（自检）
OR D1148.08  ; #3腔体机构开#3腔抽气阀（标漏步）
OR D1148.12  ; #3腔体机构开始#3-1氦检（标漏步）
OR D1149.00  ; #3腔体机构开#3腔抽真空阀（标漏步）
OR D1149.04  ; #3腔体机构开始#3-2氦检（标漏步）
ANDLD
DIFU(013) 303.06  ; #3腔体抽真空阀开[Pls]
LD TR0
LD 303.06  ; #3腔体抽真空阀开[Pls]
OR 403.06  ; #3腔体抽真空阀开[M]
ANDLD
ANDNOT 313.06  ; #3腔体抽真空阀关[Pls]
ANDNOT 822.02  ; #3腔体抽真空阀开到位标志
AND 822.09  ; #3腔体破真空阀关到位标志
AND 834.01  ; #4腔体抽真空阀关到位标志[0000.01]
AND 821.09  ; #2腔体抽真空阀关到位标志
AND 820.15  ; #1腔体抽真空阀关到位标志
AND 824.09  ; #3-1电池注氦阀关到位标志
AND 824.11  ; #3-2电池注氦阀关到位标志
AND 803.02  ; #3腔体顶伸气缸上升位标志[0003.02]
ANDNOT 803.03  ; #3腔体顶伸气缸下降位标志[0003.03]
LD 802.14  ; #3腔体平移一级气缸缩回位标志[0002.14]
AND 803.01  ; #3腔体平移二级气缸伸出位标志[0003.01]
ANDNOT 802.15  ; #3腔体平移一级气缸伸出位标志[0002.15]
ANDNOT 803.00  ; #3腔体平移二级气缸缩回位标志[0003.00]
LD 802.15  ; #3腔体平移一级气缸伸出位标志[0002.15]
AND 803.00  ; #3腔体平移二级气缸缩回位标志[0003.00]
ANDNOT 802.14  ; #3腔体平移一级气缸缩回位标志[0002.14]
ANDNOT 803.01  ; #3腔体平移二级气缸伸出位标志[0003.01]
ORLD
ANDLD
OUT 403.06  ; #3腔体抽真空阀开[M]
LD TR0
LD 713.06  ; #3腔体抽真空阀关[SW]
OR D1137.01  ; #3腔体关闭除破真空阀以外全部阀门（复位）
OR D1145.10  ; #3腔体关抽真空阀（自检）
OR D1148.09  ; #3腔体机构关#3腔体抽气阀（标漏步）
OR T2187  ; #3-1开氦检阀前抽气阀关延时（标漏）
OR D1149.01  ; #3腔体机构关#3腔抽真空阀（标漏步）
OR T2487  ; #3-2开氦检阀前抽气阀关延时（标漏）
ANDLD
DIFU(013) 313.06  ; #3腔体抽真空阀关[Pls]
LD TR0
LD 313.06  ; #3腔体抽真空阀关[Pls]
OR 413.06  ; #3腔体抽真空阀关[M]
ANDLD
ANDNOT 303.06  ; #3腔体抽真空阀开[Pls]
ANDNOT 822.03  ; #3腔体抽真空阀关到位标志
OUT 413.06  ; #3腔体抽真空阀关[M]

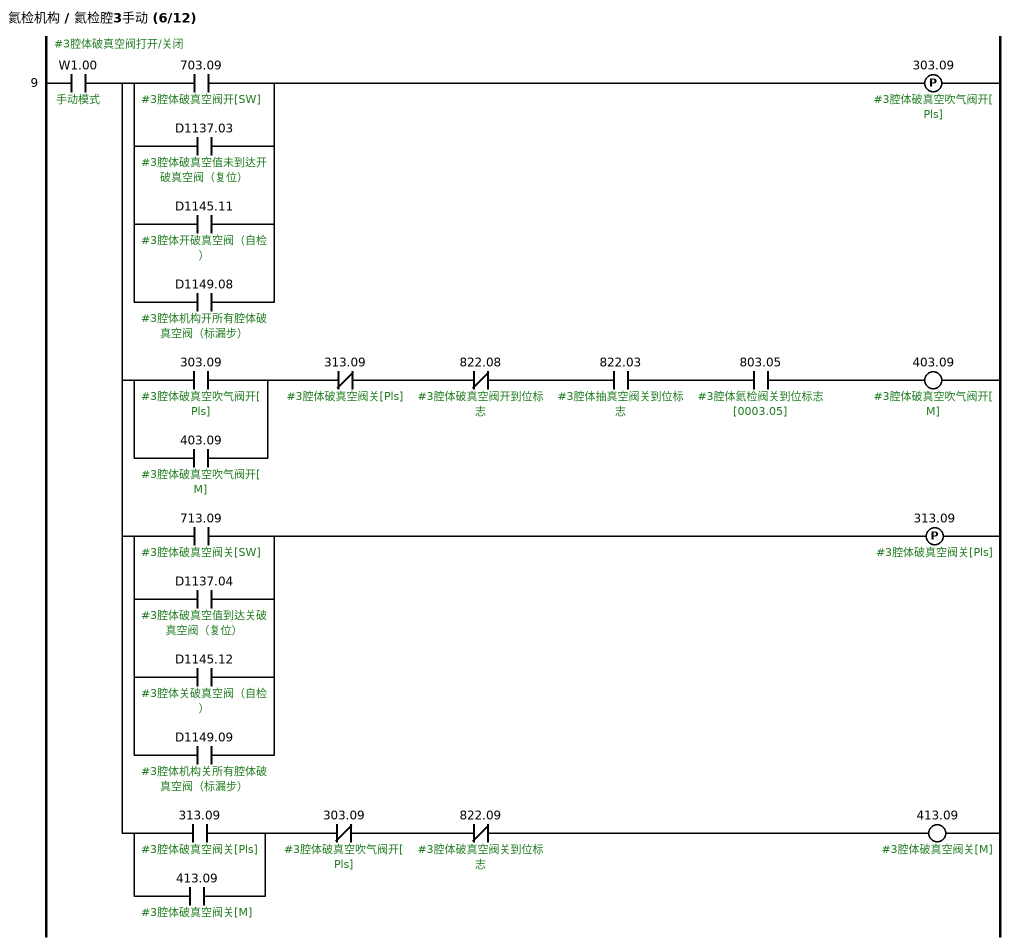
; rung 9: #3腔体破真空阀打开/关闭
LD W1.00  ; 手动模式
OUT TR0
LD 703.09  ; #3腔体破真空阀开[SW]
OR D1137.03  ; #3腔体破真空值未到达开破真空阀（复位）
OR D1145.11  ; #3腔体开破真空阀（自检）
OR D1149.08  ; #3腔体机构开所有腔体破真空阀（标漏步）
ANDLD
DIFU(013) 303.09  ; #3腔体破真空吹气阀开[Pls]
LD TR0
LD 303.09  ; #3腔体破真空吹气阀开[Pls]
OR 403.09  ; #3腔体破真空吹气阀开[M]
ANDLD
ANDNOT 313.09  ; #3腔体破真空阀关[Pls]
ANDNOT 822.08  ; #3腔体破真空阀开到位标志
AND 822.03  ; #3腔体抽真空阀关到位标志
AND 803.05  ; #3腔体氦检阀关到位标志[0003.05]
OUT 403.09  ; #3腔体破真空吹气阀开[M]
LD TR0
LD 713.09  ; #3腔体破真空阀关[SW]
OR D1137.04  ; #3腔体破真空值到达关破真空阀（复位）
OR D1145.12  ; #3腔体关破真空阀（自检）
OR D1149.09  ; #3腔体机构关所有腔体破真空阀（标漏步）
ANDLD
DIFU(013) 313.09  ; #3腔体破真空阀关[Pls]
LD TR0
LD 313.09  ; #3腔体破真空阀关[Pls]
OR 413.09  ; #3腔体破真空阀关[M]
ANDLD
ANDNOT 303.09  ; #3腔体破真空吹气阀开[Pls]
ANDNOT 822.09  ; #3腔体破真空阀关到位标志
OUT 413.09  ; #3腔体破真空阀关[M]

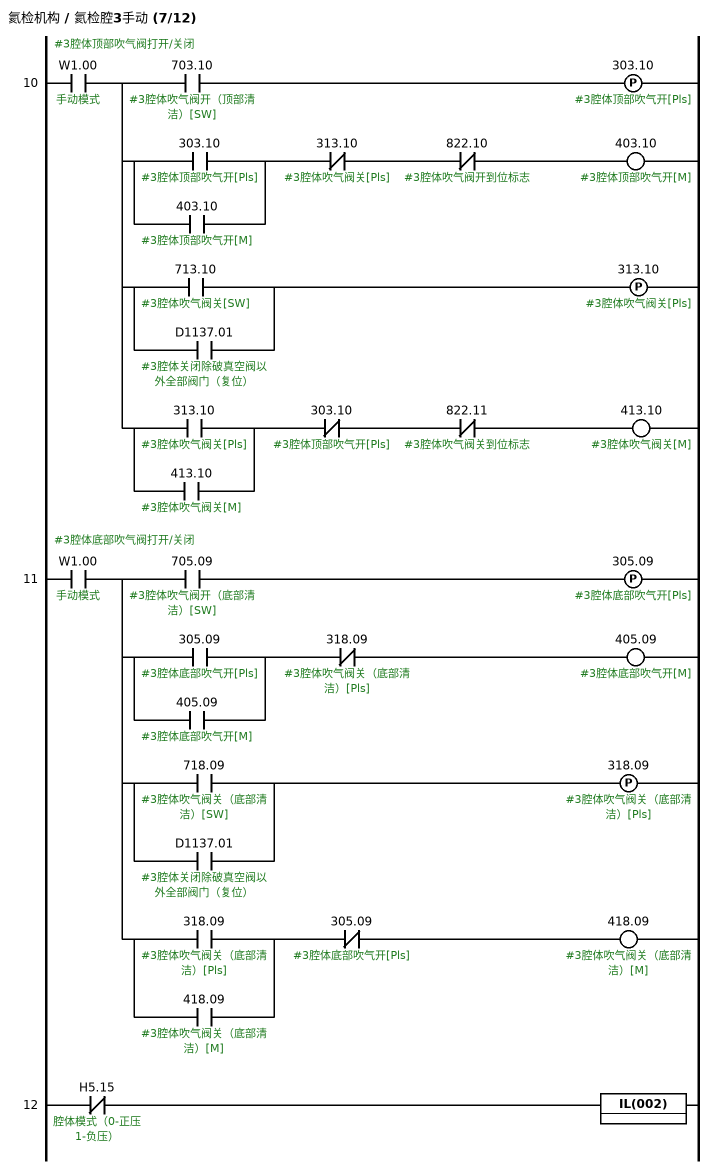
; rung 10: #3腔体顶部吹气阀打开/关闭
LD W1.00  ; 手动模式
OUT TR0
AND 703.10  ; #3腔体吹气阀开（顶部清洁）[SW]
DIFU(013) 303.10  ; #3腔体顶部吹气开[Pls]
LD TR0
LD 303.10  ; #3腔体顶部吹气开[Pls]
OR 403.10  ; #3腔体顶部吹气开[M]
ANDLD
ANDNOT 313.10  ; #3腔体吹气阀关[Pls]
ANDNOT 822.10  ; #3腔体吹气阀开到位标志
OUT 403.10  ; #3腔体顶部吹气开[M]
LD TR0
LD 713.10  ; #3腔体吹气阀关[SW]
OR D1137.01  ; #3腔体关闭除破真空阀以外全部阀门（复位）
ANDLD
DIFU(013) 313.10  ; #3腔体吹气阀关[Pls]
LD TR0
LD 313.10  ; #3腔体吹气阀关[Pls]
OR 413.10  ; #3腔体吹气阀关[M]
ANDLD
ANDNOT 303.10  ; #3腔体顶部吹气开[Pls]
ANDNOT 822.11  ; #3腔体吹气阀关到位标志
OUT 413.10  ; #3腔体吹气阀关[M]
; rung 11: #3腔体底部吹气阀打开/关闭
LD W1.00  ; 手动模式
OUT TR0
AND 705.09  ; #3腔体吹气阀开（底部清洁）[SW]
DIFU(013) 305.09  ; #3腔体底部吹气开[Pls]
LD TR0
LD 305.09  ; #3腔体底部吹气开[Pls]
OR 405.09  ; #3腔体底部吹气开[M]
ANDLD
ANDNOT 318.09  ; #3腔体吹气阀关（底部清洁）[Pls]
OUT 405.09  ; #3腔体底部吹气开[M]
LD TR0
LD 718.09  ; #3腔体吹气阀关（底部清洁）[SW]
OR D1137.01  ; #3腔体关闭除破真空阀以外全部阀门（复位）
ANDLD
DIFU(013) 318.09  ; #3腔体吹气阀关（底部清洁）[Pls]
LD TR0
LD 318.09  ; #3腔体吹气阀关（底部清洁）[Pls]
OR 418.09  ; #3腔体吹气阀关（底部清洁）[M]
ANDLD
ANDNOT 305.09  ; #3腔体底部吹气开[Pls]
OUT 418.09  ; #3腔体吹气阀关（底部清洁）[M]
; rung 12
LDNOT H5.15  ; 腔体模式（0-正压 1-负压）
IL(002)

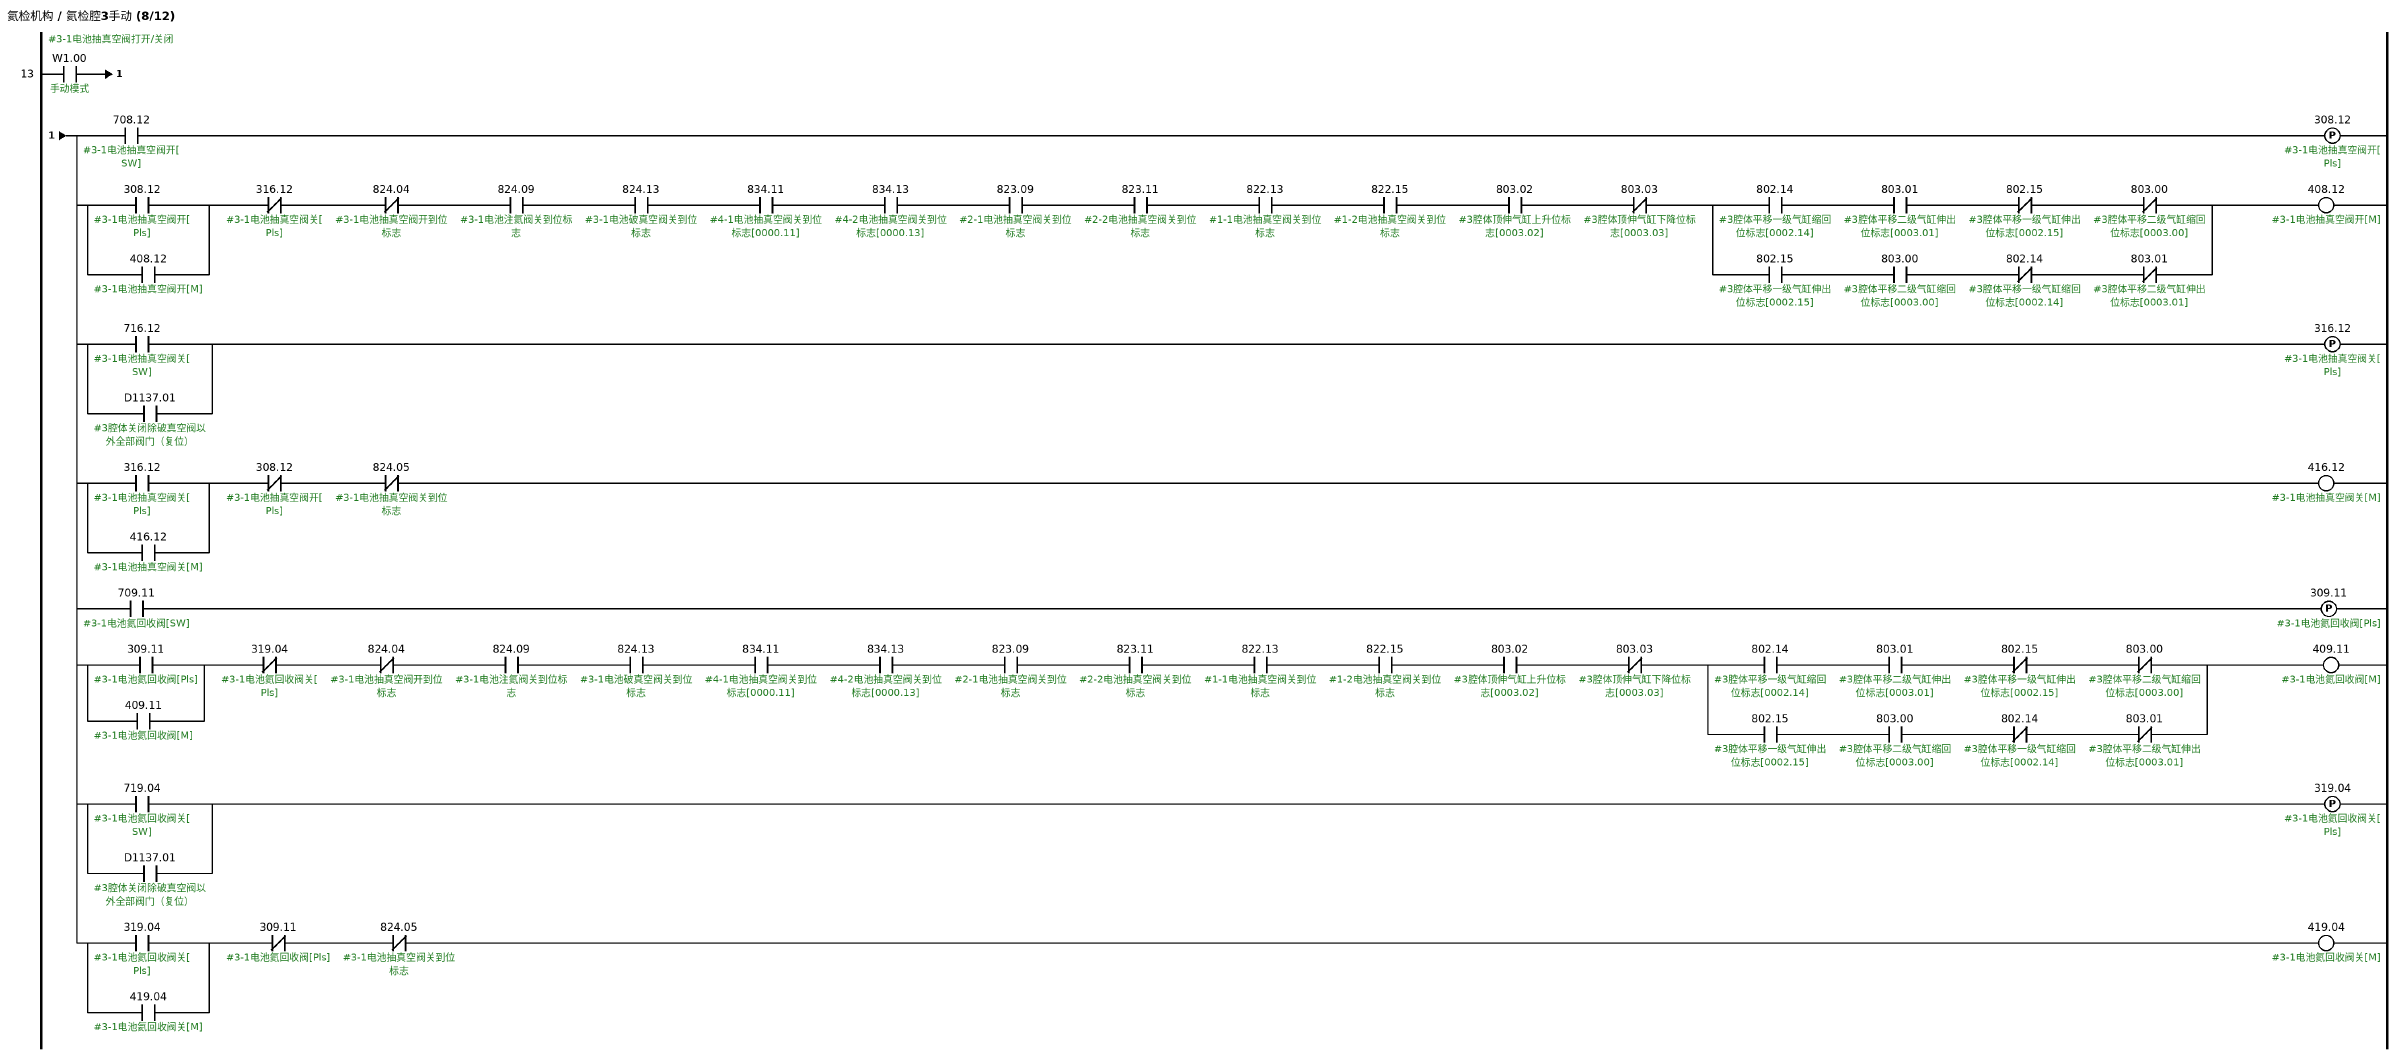
; rung 13: #3-1电池抽真空阀打开/关闭
LD W1.00  ; 手动模式
OUT TR0
AND 708.12  ; #3-1电池抽真空阀开[SW]
DIFU(013) 308.12  ; #3-1电池抽真空阀开[Pls]
LD TR0
LD 308.12  ; #3-1电池抽真空阀开[Pls]
OR 408.12  ; #3-1电池抽真空阀开[M]
ANDLD
ANDNOT 316.12  ; #3-1电池抽真空阀关[Pls]
ANDNOT 824.04  ; #3-1电池抽真空阀开到位标志
AND 824.09  ; #3-1电池注氦阀关到位标志
AND 824.13  ; #3-1电池破真空阀关到位标志
AND 834.11  ; #4-1电池抽真空阀关到位标志[0000.11]
AND 834.13  ; #4-2电池抽真空阀关到位标志[0000.13]
AND 823.09  ; #2-1电池抽真空阀关到位标志
AND 823.11  ; #2-2电池抽真空阀关到位标志
AND 822.13  ; #1-1电池抽真空阀关到位标志
AND 822.15  ; #1-2电池抽真空阀关到位标志
AND 803.02  ; #3腔体顶伸气缸上升位标志[0003.02]
ANDNOT 803.03  ; #3腔体顶伸气缸下降位标志[0003.03]
LD 802.14  ; #3腔体平移一级气缸缩回位标志[0002.14]
AND 803.01  ; #3腔体平移二级气缸伸出位标志[0003.01]
ANDNOT 802.15  ; #3腔体平移一级气缸伸出位标志[0002.15]
ANDNOT 803.00  ; #3腔体平移二级气缸缩回位标志[0003.00]
LD 802.15  ; #3腔体平移一级气缸伸出位标志[0002.15]
AND 803.00  ; #3腔体平移二级气缸缩回位标志[0003.00]
ANDNOT 802.14  ; #3腔体平移一级气缸缩回位标志[0002.14]
ANDNOT 803.01  ; #3腔体平移二级气缸伸出位标志[0003.01]
ORLD
ANDLD
OUT 408.12  ; #3-1电池抽真空阀开[M]
LD TR0
LD 716.12  ; #3-1电池抽真空阀关[SW]
OR D1137.01  ; #3腔体关闭除破真空阀以外全部阀门（复位）
ANDLD
DIFU(013) 316.12  ; #3-1电池抽真空阀关[Pls]
LD TR0
LD 316.12  ; #3-1电池抽真空阀关[Pls]
OR 416.12  ; #3-1电池抽真空阀关[M]
ANDLD
ANDNOT 308.12  ; #3-1电池抽真空阀开[Pls]
ANDNOT 824.05  ; #3-1电池抽真空阀关到位标志
OUT 416.12  ; #3-1电池抽真空阀关[M]
LD TR0
AND 709.11  ; #3-1电池氦回收阀[SW]
DIFU(013) 309.11  ; #3-1电池氦回收阀[Pls]
LD TR0
LD 309.11  ; #3-1电池氦回收阀[Pls]
OR 409.11  ; #3-1电池氦回收阀[M]
ANDLD
ANDNOT 319.04  ; #3-1电池氦回收阀关[Pls]
ANDNOT 824.04  ; #3-1电池抽真空阀开到位标志
AND 824.09  ; #3-1电池注氦阀关到位标志
AND 824.13  ; #3-1电池破真空阀关到位标志
AND 834.11  ; #4-1电池抽真空阀关到位标志[0000.11]
AND 834.13  ; #4-2电池抽真空阀关到位标志[0000.13]
AND 823.09  ; #2-1电池抽真空阀关到位标志
AND 823.11  ; #2-2电池抽真空阀关到位标志
AND 822.13  ; #1-1电池抽真空阀关到位标志
AND 822.15  ; #1-2电池抽真空阀关到位标志
AND 803.02  ; #3腔体顶伸气缸上升位标志[0003.02]
ANDNOT 803.03  ; #3腔体顶伸气缸下降位标志[0003.03]
LD 802.14  ; #3腔体平移一级气缸缩回位标志[0002.14]
AND 803.01  ; #3腔体平移二级气缸伸出位标志[0003.01]
ANDNOT 802.15  ; #3腔体平移一级气缸伸出位标志[0002.15]
ANDNOT 803.00  ; #3腔体平移二级气缸缩回位标志[0003.00]
LD 802.15  ; #3腔体平移一级气缸伸出位标志[0002.15]
AND 803.00  ; #3腔体平移二级气缸缩回位标志[0003.00]
ANDNOT 802.14  ; #3腔体平移一级气缸缩回位标志[0002.14]
ANDNOT 803.01  ; #3腔体平移二级气缸伸出位标志[0003.01]
ORLD
ANDLD
OUT 409.11  ; #3-1电池氦回收阀[M]
LD TR0
LD 719.04  ; #3-1电池氦回收阀关[SW]
OR D1137.01  ; #3腔体关闭除破真空阀以外全部阀门（复位）
ANDLD
DIFU(013) 319.04  ; #3-1电池氦回收阀关[Pls]
LD TR0
LD 319.04  ; #3-1电池氦回收阀关[Pls]
OR 419.04  ; #3-1电池氦回收阀关[M]
ANDLD
ANDNOT 309.11  ; #3-1电池氦回收阀[Pls]
ANDNOT 824.05  ; #3-1电池抽真空阀关到位标志
OUT 419.04  ; #3-1电池氦回收阀关[M]

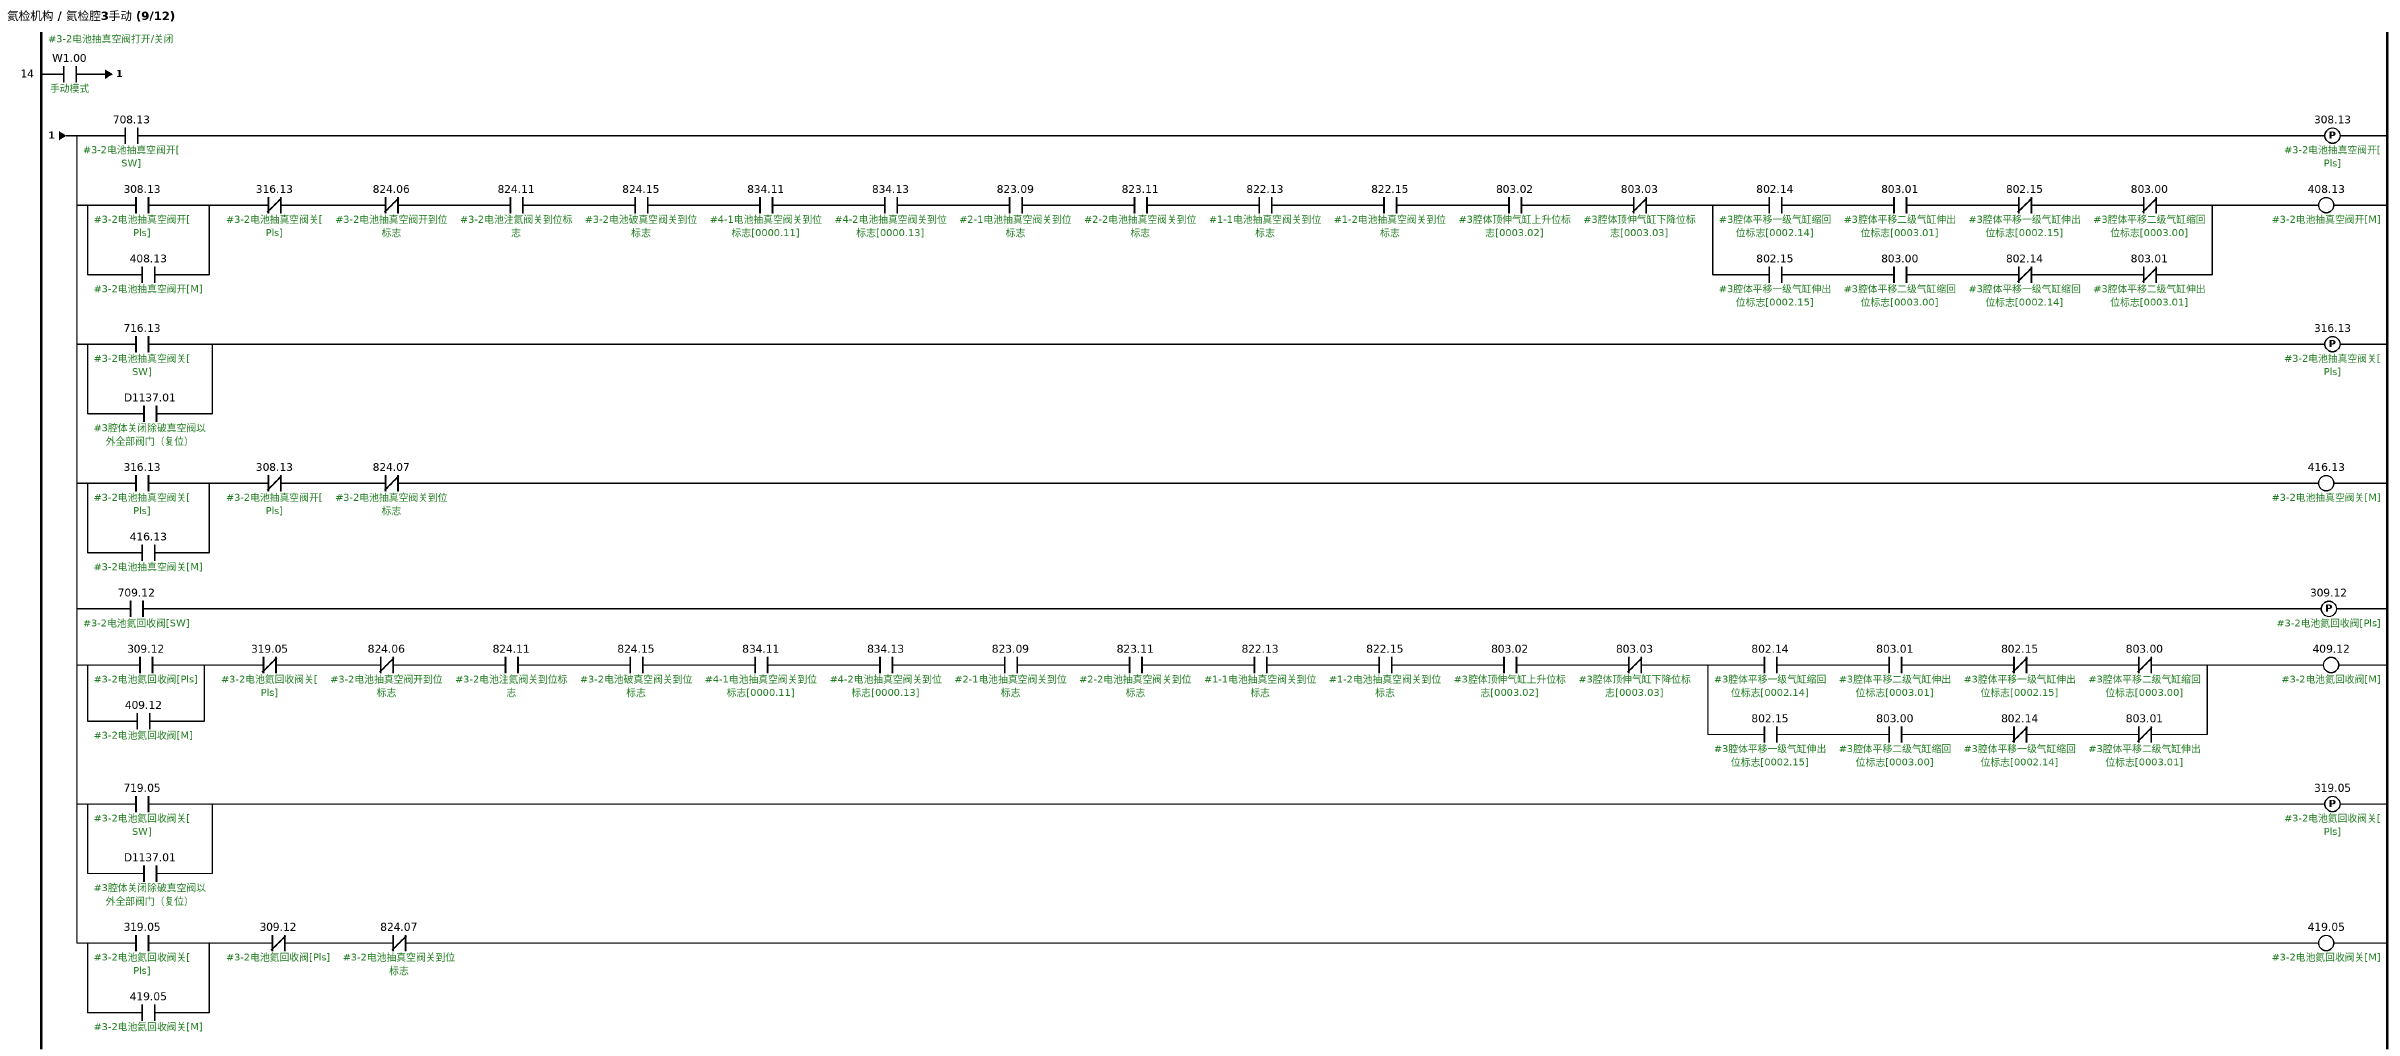
; rung 14: #3-2电池抽真空阀打开/关闭
LD W1.00  ; 手动模式
OUT TR0
AND 708.13  ; #3-2电池抽真空阀开[SW]
DIFU(013) 308.13  ; #3-2电池抽真空阀开[Pls]
LD TR0
LD 308.13  ; #3-2电池抽真空阀开[Pls]
OR 408.13  ; #3-2电池抽真空阀开[M]
ANDLD
ANDNOT 316.13  ; #3-2电池抽真空阀关[Pls]
ANDNOT 824.06  ; #3-2电池抽真空阀开到位标志
AND 824.11  ; #3-2电池注氦阀关到位标志
AND 824.15  ; #3-2电池破真空阀关到位标志
AND 834.11  ; #4-1电池抽真空阀关到位标志[0000.11]
AND 834.13  ; #4-2电池抽真空阀关到位标志[0000.13]
AND 823.09  ; #2-1电池抽真空阀关到位标志
AND 823.11  ; #2-2电池抽真空阀关到位标志
AND 822.13  ; #1-1电池抽真空阀关到位标志
AND 822.15  ; #1-2电池抽真空阀关到位标志
AND 803.02  ; #3腔体顶伸气缸上升位标志[0003.02]
ANDNOT 803.03  ; #3腔体顶伸气缸下降位标志[0003.03]
LD 802.14  ; #3腔体平移一级气缸缩回位标志[0002.14]
AND 803.01  ; #3腔体平移二级气缸伸出位标志[0003.01]
ANDNOT 802.15  ; #3腔体平移一级气缸伸出位标志[0002.15]
ANDNOT 803.00  ; #3腔体平移二级气缸缩回位标志[0003.00]
LD 802.15  ; #3腔体平移一级气缸伸出位标志[0002.15]
AND 803.00  ; #3腔体平移二级气缸缩回位标志[0003.00]
ANDNOT 802.14  ; #3腔体平移一级气缸缩回位标志[0002.14]
ANDNOT 803.01  ; #3腔体平移二级气缸伸出位标志[0003.01]
ORLD
ANDLD
OUT 408.13  ; #3-2电池抽真空阀开[M]
LD TR0
LD 716.13  ; #3-2电池抽真空阀关[SW]
OR D1137.01  ; #3腔体关闭除破真空阀以外全部阀门（复位）
ANDLD
DIFU(013) 316.13  ; #3-2电池抽真空阀关[Pls]
LD TR0
LD 316.13  ; #3-2电池抽真空阀关[Pls]
OR 416.13  ; #3-2电池抽真空阀关[M]
ANDLD
ANDNOT 308.13  ; #3-2电池抽真空阀开[Pls]
ANDNOT 824.07  ; #3-2电池抽真空阀关到位标志
OUT 416.13  ; #3-2电池抽真空阀关[M]
LD TR0
AND 709.12  ; #3-2电池氦回收阀[SW]
DIFU(013) 309.12  ; #3-2电池氦回收阀[Pls]
LD TR0
LD 309.12  ; #3-2电池氦回收阀[Pls]
OR 409.12  ; #3-2电池氦回收阀[M]
ANDLD
ANDNOT 319.05  ; #3-2电池氦回收阀关[Pls]
ANDNOT 824.06  ; #3-2电池抽真空阀开到位标志
AND 824.11  ; #3-2电池注氦阀关到位标志
AND 824.15  ; #3-2电池破真空阀关到位标志
AND 834.11  ; #4-1电池抽真空阀关到位标志[0000.11]
AND 834.13  ; #4-2电池抽真空阀关到位标志[0000.13]
AND 823.09  ; #2-1电池抽真空阀关到位标志
AND 823.11  ; #2-2电池抽真空阀关到位标志
AND 822.13  ; #1-1电池抽真空阀关到位标志
AND 822.15  ; #1-2电池抽真空阀关到位标志
AND 803.02  ; #3腔体顶伸气缸上升位标志[0003.02]
ANDNOT 803.03  ; #3腔体顶伸气缸下降位标志[0003.03]
LD 802.14  ; #3腔体平移一级气缸缩回位标志[0002.14]
AND 803.01  ; #3腔体平移二级气缸伸出位标志[0003.01]
ANDNOT 802.15  ; #3腔体平移一级气缸伸出位标志[0002.15]
ANDNOT 803.00  ; #3腔体平移二级气缸缩回位标志[0003.00]
LD 802.15  ; #3腔体平移一级气缸伸出位标志[0002.15]
AND 803.00  ; #3腔体平移二级气缸缩回位标志[0003.00]
ANDNOT 802.14  ; #3腔体平移一级气缸缩回位标志[0002.14]
ANDNOT 803.01  ; #3腔体平移二级气缸伸出位标志[0003.01]
ORLD
ANDLD
OUT 409.12  ; #3-2电池氦回收阀[M]
LD TR0
LD 719.05  ; #3-2电池氦回收阀关[SW]
OR D1137.01  ; #3腔体关闭除破真空阀以外全部阀门（复位）
ANDLD
DIFU(013) 319.05  ; #3-2电池氦回收阀关[Pls]
LD TR0
LD 319.05  ; #3-2电池氦回收阀关[Pls]
OR 419.05  ; #3-2电池氦回收阀关[M]
ANDLD
ANDNOT 309.12  ; #3-2电池氦回收阀[Pls]
ANDNOT 824.07  ; #3-2电池抽真空阀关到位标志
OUT 419.05  ; #3-2电池氦回收阀关[M]

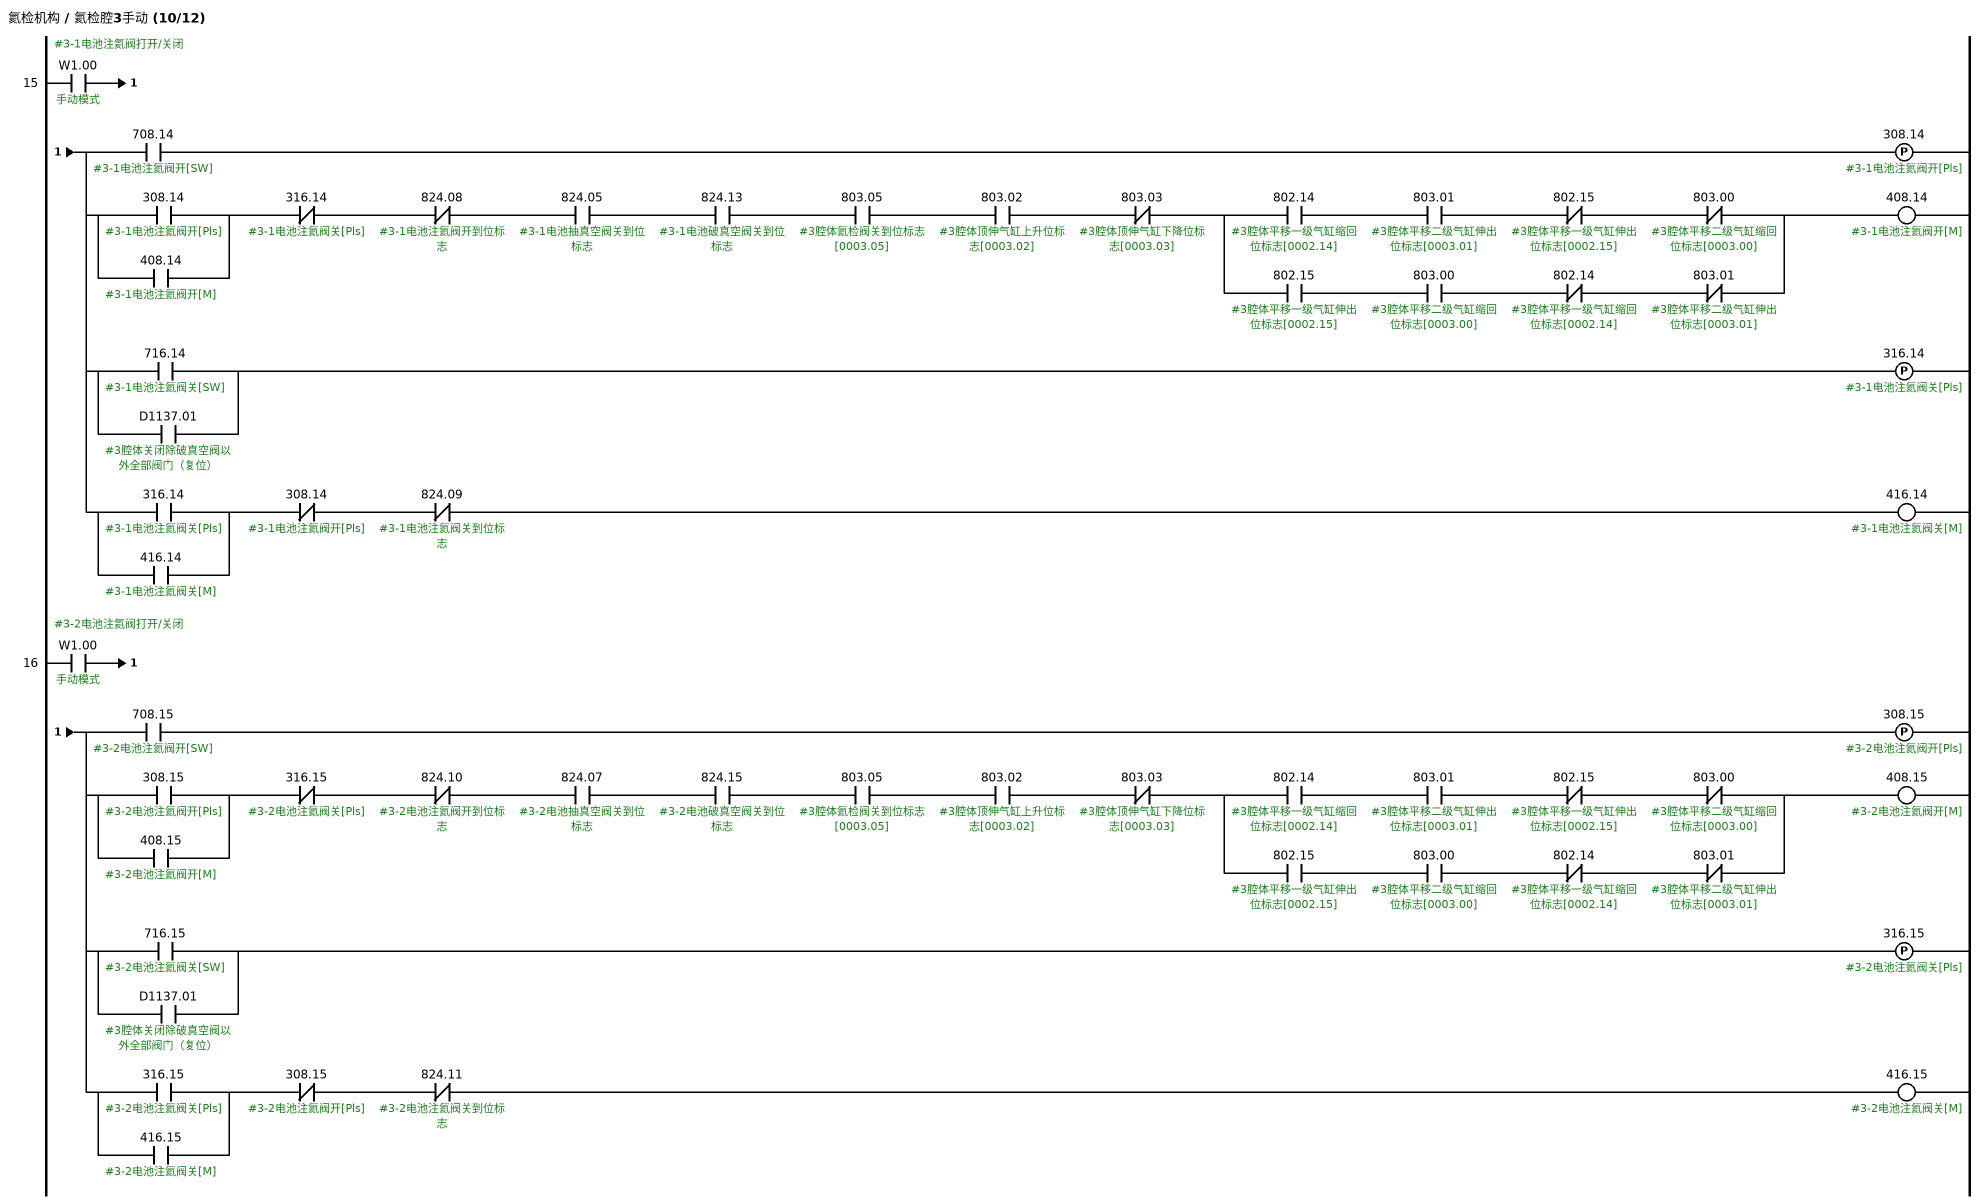
; rung 15: #3-1电池注氦阀打开/关闭
LD W1.00  ; 手动模式
OUT TR0
AND 708.14  ; #3-1电池注氦阀开[SW]
DIFU(013) 308.14  ; #3-1电池注氦阀开[Pls]
LD TR0
LD 308.14  ; #3-1电池注氦阀开[Pls]
OR 408.14  ; #3-1电池注氦阀开[M]
ANDLD
ANDNOT 316.14  ; #3-1电池注氦阀关[Pls]
ANDNOT 824.08  ; #3-1电池注氦阀开到位标志
AND 824.05  ; #3-1电池抽真空阀关到位标志
AND 824.13  ; #3-1电池破真空阀关到位标志
AND 803.05  ; #3腔体氦检阀关到位标志[0003.05]
AND 803.02  ; #3腔体顶伸气缸上升位标志[0003.02]
ANDNOT 803.03  ; #3腔体顶伸气缸下降位标志[0003.03]
LD 802.14  ; #3腔体平移一级气缸缩回位标志[0002.14]
AND 803.01  ; #3腔体平移二级气缸伸出位标志[0003.01]
ANDNOT 802.15  ; #3腔体平移一级气缸伸出位标志[0002.15]
ANDNOT 803.00  ; #3腔体平移二级气缸缩回位标志[0003.00]
LD 802.15  ; #3腔体平移一级气缸伸出位标志[0002.15]
AND 803.00  ; #3腔体平移二级气缸缩回位标志[0003.00]
ANDNOT 802.14  ; #3腔体平移一级气缸缩回位标志[0002.14]
ANDNOT 803.01  ; #3腔体平移二级气缸伸出位标志[0003.01]
ORLD
ANDLD
OUT 408.14  ; #3-1电池注氦阀开[M]
LD TR0
LD 716.14  ; #3-1电池注氦阀关[SW]
OR D1137.01  ; #3腔体关闭除破真空阀以外全部阀门（复位）
ANDLD
DIFU(013) 316.14  ; #3-1电池注氦阀关[Pls]
LD TR0
LD 316.14  ; #3-1电池注氦阀关[Pls]
OR 416.14  ; #3-1电池注氦阀关[M]
ANDLD
ANDNOT 308.14  ; #3-1电池注氦阀开[Pls]
ANDNOT 824.09  ; #3-1电池注氦阀关到位标志
OUT 416.14  ; #3-1电池注氦阀关[M]
; rung 16: #3-2电池注氦阀打开/关闭
LD W1.00  ; 手动模式
OUT TR0
AND 708.15  ; #3-2电池注氦阀开[SW]
DIFU(013) 308.15  ; #3-2电池注氦阀开[Pls]
LD TR0
LD 308.15  ; #3-2电池注氦阀开[Pls]
OR 408.15  ; #3-2电池注氦阀开[M]
ANDLD
ANDNOT 316.15  ; #3-2电池注氦阀关[Pls]
ANDNOT 824.10  ; #3-2电池注氦阀开到位标志
AND 824.07  ; #3-2电池抽真空阀关到位标志
AND 824.15  ; #3-2电池破真空阀关到位标志
AND 803.05  ; #3腔体氦检阀关到位标志[0003.05]
AND 803.02  ; #3腔体顶伸气缸上升位标志[0003.02]
ANDNOT 803.03  ; #3腔体顶伸气缸下降位标志[0003.03]
LD 802.14  ; #3腔体平移一级气缸缩回位标志[0002.14]
AND 803.01  ; #3腔体平移二级气缸伸出位标志[0003.01]
ANDNOT 802.15  ; #3腔体平移一级气缸伸出位标志[0002.15]
ANDNOT 803.00  ; #3腔体平移二级气缸缩回位标志[0003.00]
LD 802.15  ; #3腔体平移一级气缸伸出位标志[0002.15]
AND 803.00  ; #3腔体平移二级气缸缩回位标志[0003.00]
ANDNOT 802.14  ; #3腔体平移一级气缸缩回位标志[0002.14]
ANDNOT 803.01  ; #3腔体平移二级气缸伸出位标志[0003.01]
ORLD
ANDLD
OUT 408.15  ; #3-2电池注氦阀开[M]
LD TR0
LD 716.15  ; #3-2电池注氦阀关[SW]
OR D1137.01  ; #3腔体关闭除破真空阀以外全部阀门（复位）
ANDLD
DIFU(013) 316.15  ; #3-2电池注氦阀关[Pls]
LD TR0
LD 316.15  ; #3-2电池注氦阀关[Pls]
OR 416.15  ; #3-2电池注氦阀关[M]
ANDLD
ANDNOT 308.15  ; #3-2电池注氦阀开[Pls]
ANDNOT 824.11  ; #3-2电池注氦阀关到位标志
OUT 416.15  ; #3-2电池注氦阀关[M]

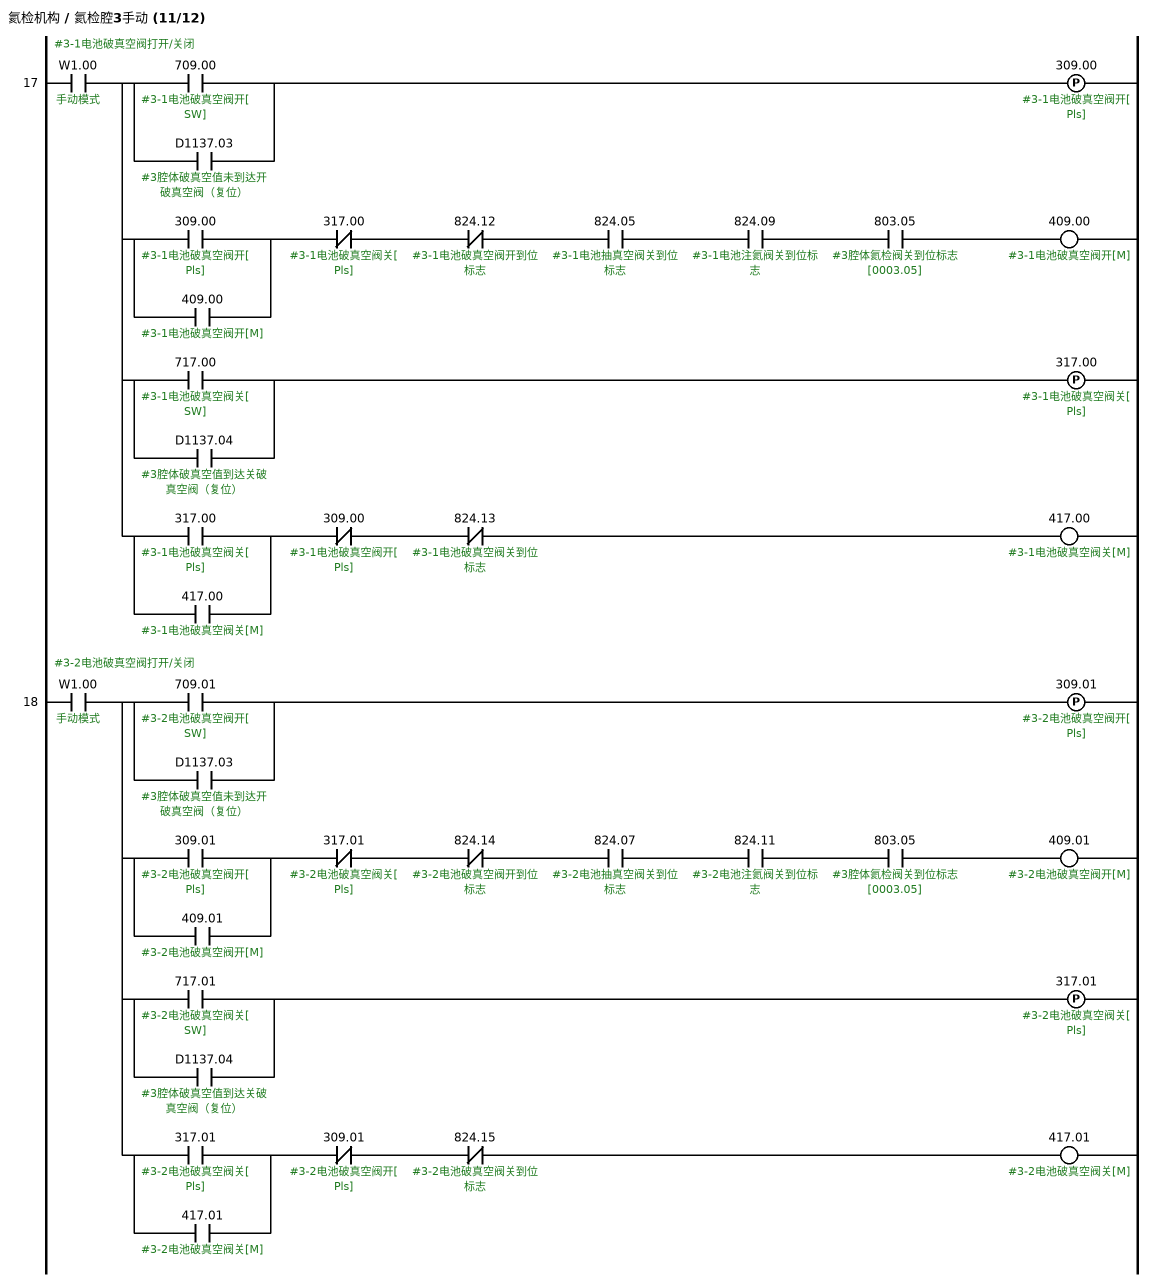
; rung 17: #3-1电池破真空阀打开/关闭
LD W1.00  ; 手动模式
OUT TR0
LD 709.00  ; #3-1电池破真空阀开[SW]
OR D1137.03  ; #3腔体破真空值未到达开破真空阀（复位）
ANDLD
DIFU(013) 309.00  ; #3-1电池破真空阀开[Pls]
LD TR0
LD 309.00  ; #3-1电池破真空阀开[Pls]
OR 409.00  ; #3-1电池破真空阀开[M]
ANDLD
ANDNOT 317.00  ; #3-1电池破真空阀关[Pls]
ANDNOT 824.12  ; #3-1电池破真空阀开到位标志
AND 824.05  ; #3-1电池抽真空阀关到位标志
AND 824.09  ; #3-1电池注氦阀关到位标志
AND 803.05  ; #3腔体氦检阀关到位标志[0003.05]
OUT 409.00  ; #3-1电池破真空阀开[M]
LD TR0
LD 717.00  ; #3-1电池破真空阀关[SW]
OR D1137.04  ; #3腔体破真空值到达关破真空阀（复位）
ANDLD
DIFU(013) 317.00  ; #3-1电池破真空阀关[Pls]
LD TR0
LD 317.00  ; #3-1电池破真空阀关[Pls]
OR 417.00  ; #3-1电池破真空阀关[M]
ANDLD
ANDNOT 309.00  ; #3-1电池破真空阀开[Pls]
ANDNOT 824.13  ; #3-1电池破真空阀关到位标志
OUT 417.00  ; #3-1电池破真空阀关[M]
; rung 18: #3-2电池破真空阀打开/关闭
LD W1.00  ; 手动模式
OUT TR0
LD 709.01  ; #3-2电池破真空阀开[SW]
OR D1137.03  ; #3腔体破真空值未到达开破真空阀（复位）
ANDLD
DIFU(013) 309.01  ; #3-2电池破真空阀开[Pls]
LD TR0
LD 309.01  ; #3-2电池破真空阀开[Pls]
OR 409.01  ; #3-2电池破真空阀开[M]
ANDLD
ANDNOT 317.01  ; #3-2电池破真空阀关[Pls]
ANDNOT 824.14  ; #3-2电池破真空阀开到位标志
AND 824.07  ; #3-2电池抽真空阀关到位标志
AND 824.11  ; #3-2电池注氦阀关到位标志
AND 803.05  ; #3腔体氦检阀关到位标志[0003.05]
OUT 409.01  ; #3-2电池破真空阀开[M]
LD TR0
LD 717.01  ; #3-2电池破真空阀关[SW]
OR D1137.04  ; #3腔体破真空值到达关破真空阀（复位）
ANDLD
DIFU(013) 317.01  ; #3-2电池破真空阀关[Pls]
LD TR0
LD 317.01  ; #3-2电池破真空阀关[Pls]
OR 417.01  ; #3-2电池破真空阀关[M]
ANDLD
ANDNOT 309.01  ; #3-2电池破真空阀开[Pls]
ANDNOT 824.15  ; #3-2电池破真空阀关到位标志
OUT 417.01  ; #3-2电池破真空阀关[M]

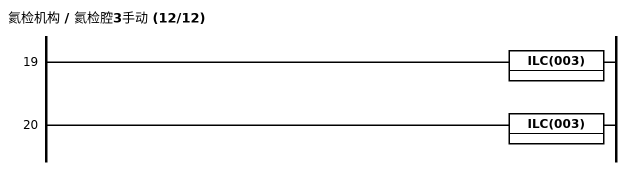
; rung 19
ILC(003)
; rung 20
ILC(003)

### Section 氦检腔4手动

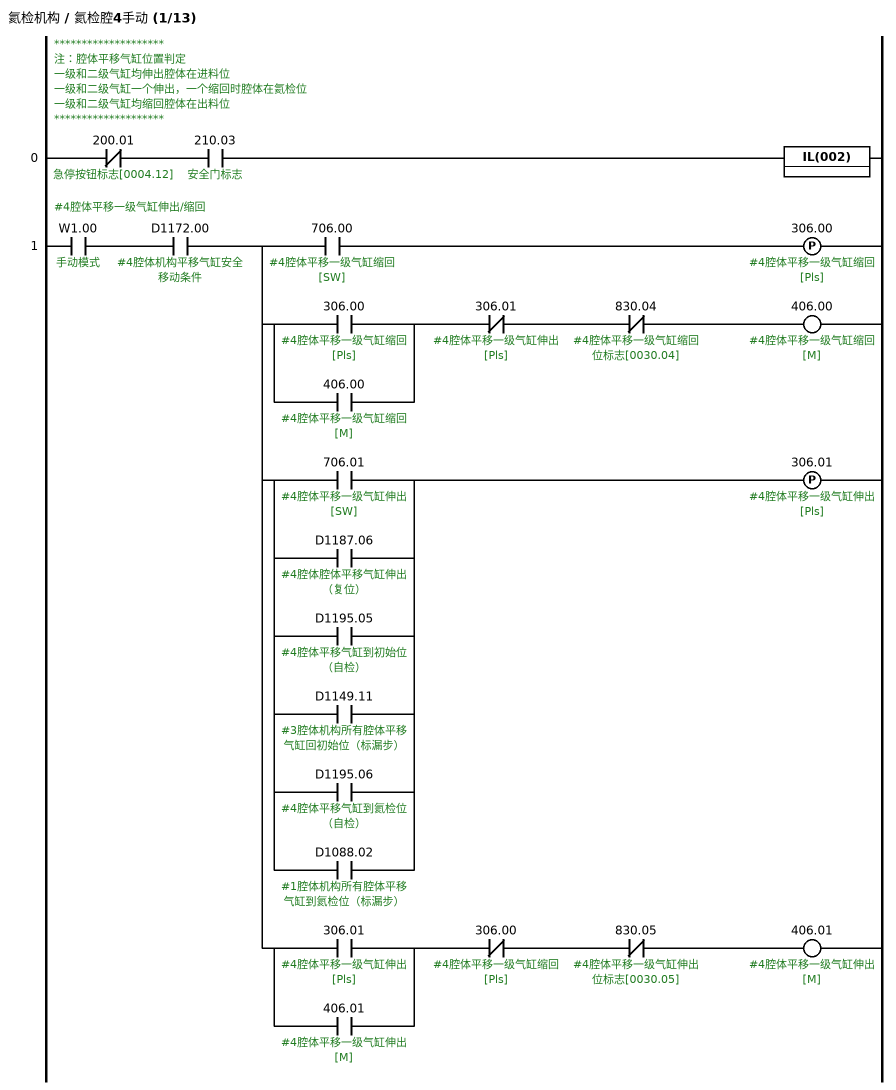
; rung 0: ******************** / 注：腔体平移气缸位置判定 / 一级和二级气缸均伸出腔体在进料位 / 一级和二级气缸一个伸出，一个缩回时腔体在氦检位 / 一级和二级气缸均缩回腔体在出料位 / ********************
LDNOT 200.01  ; 急停按钮标志[0004.12]
AND 210.03  ; 安全门标志
IL(002)
; rung 1: #4腔体平移一级气缸伸出/缩回
LD W1.00  ; 手动模式
AND D1172.00  ; #4腔体机构平移气缸安全移动条件
OUT TR0
AND 706.00  ; #4腔体平移一级气缸缩回[SW]
DIFU(013) 306.00  ; #4腔体平移一级气缸缩回[Pls]
LD TR0
LD 306.00  ; #4腔体平移一级气缸缩回[Pls]
OR 406.00  ; #4腔体平移一级气缸缩回[M]
ANDLD
ANDNOT 306.01  ; #4腔体平移一级气缸伸出[Pls]
ANDNOT 830.04  ; #4腔体平移一级气缸缩回位标志[0030.04]
OUT 406.00  ; #4腔体平移一级气缸缩回[M]
LD TR0
LD 706.01  ; #4腔体平移一级气缸伸出[SW]
OR D1187.06  ; #4腔体腔体平移气缸伸出（复位）
OR D1195.05  ; #4腔体平移气缸到初始位（自检）
OR D1149.11  ; #3腔体机构所有腔体平移气缸回初始位（标漏步）
OR D1195.06  ; #4腔体平移气缸到氦检位（自检）
OR D1088.02  ; #1腔体机构所有腔体平移气缸到氦检位（标漏步）
ANDLD
DIFU(013) 306.01  ; #4腔体平移一级气缸伸出[Pls]
LD TR0
LD 306.01  ; #4腔体平移一级气缸伸出[Pls]
OR 406.01  ; #4腔体平移一级气缸伸出[M]
ANDLD
ANDNOT 306.00  ; #4腔体平移一级气缸缩回[Pls]
ANDNOT 830.05  ; #4腔体平移一级气缸伸出位标志[0030.05]
OUT 406.01  ; #4腔体平移一级气缸伸出[M]

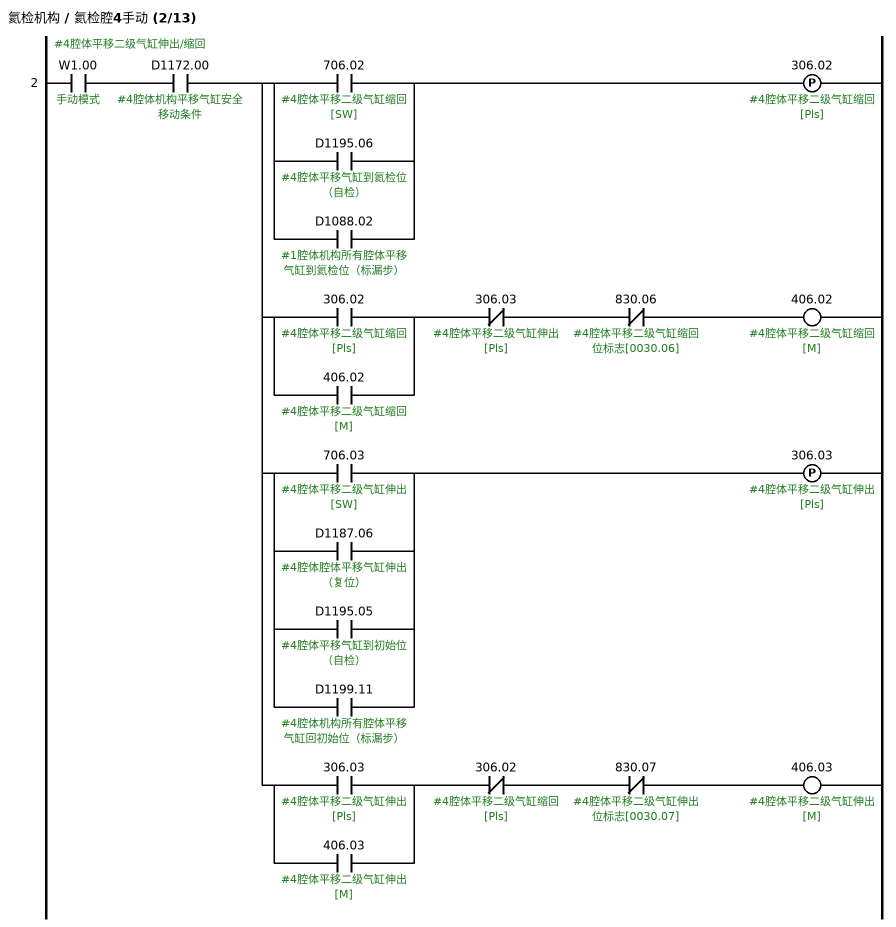
; rung 2: #4腔体平移二级气缸伸出/缩回
LD W1.00  ; 手动模式
AND D1172.00  ; #4腔体机构平移气缸安全移动条件
OUT TR0
LD 706.02  ; #4腔体平移二级气缸缩回[SW]
OR D1195.06  ; #4腔体平移气缸到氦检位（自检）
OR D1088.02  ; #1腔体机构所有腔体平移气缸到氦检位（标漏步）
ANDLD
DIFU(013) 306.02  ; #4腔体平移二级气缸缩回[Pls]
LD TR0
LD 306.02  ; #4腔体平移二级气缸缩回[Pls]
OR 406.02  ; #4腔体平移二级气缸缩回[M]
ANDLD
ANDNOT 306.03  ; #4腔体平移二级气缸伸出[Pls]
ANDNOT 830.06  ; #4腔体平移二级气缸缩回位标志[0030.06]
OUT 406.02  ; #4腔体平移二级气缸缩回[M]
LD TR0
LD 706.03  ; #4腔体平移二级气缸伸出[SW]
OR D1187.06  ; #4腔体腔体平移气缸伸出（复位）
OR D1195.05  ; #4腔体平移气缸到初始位（自检）
OR D1199.11  ; #4腔体机构所有腔体平移气缸回初始位（标漏步）
ANDLD
DIFU(013) 306.03  ; #4腔体平移二级气缸伸出[Pls]
LD TR0
LD 306.03  ; #4腔体平移二级气缸伸出[Pls]
OR 406.03  ; #4腔体平移二级气缸伸出[M]
ANDLD
ANDNOT 306.02  ; #4腔体平移二级气缸缩回[Pls]
ANDNOT 830.07  ; #4腔体平移二级气缸伸出位标志[0030.07]
OUT 406.03  ; #4腔体平移二级气缸伸出[M]

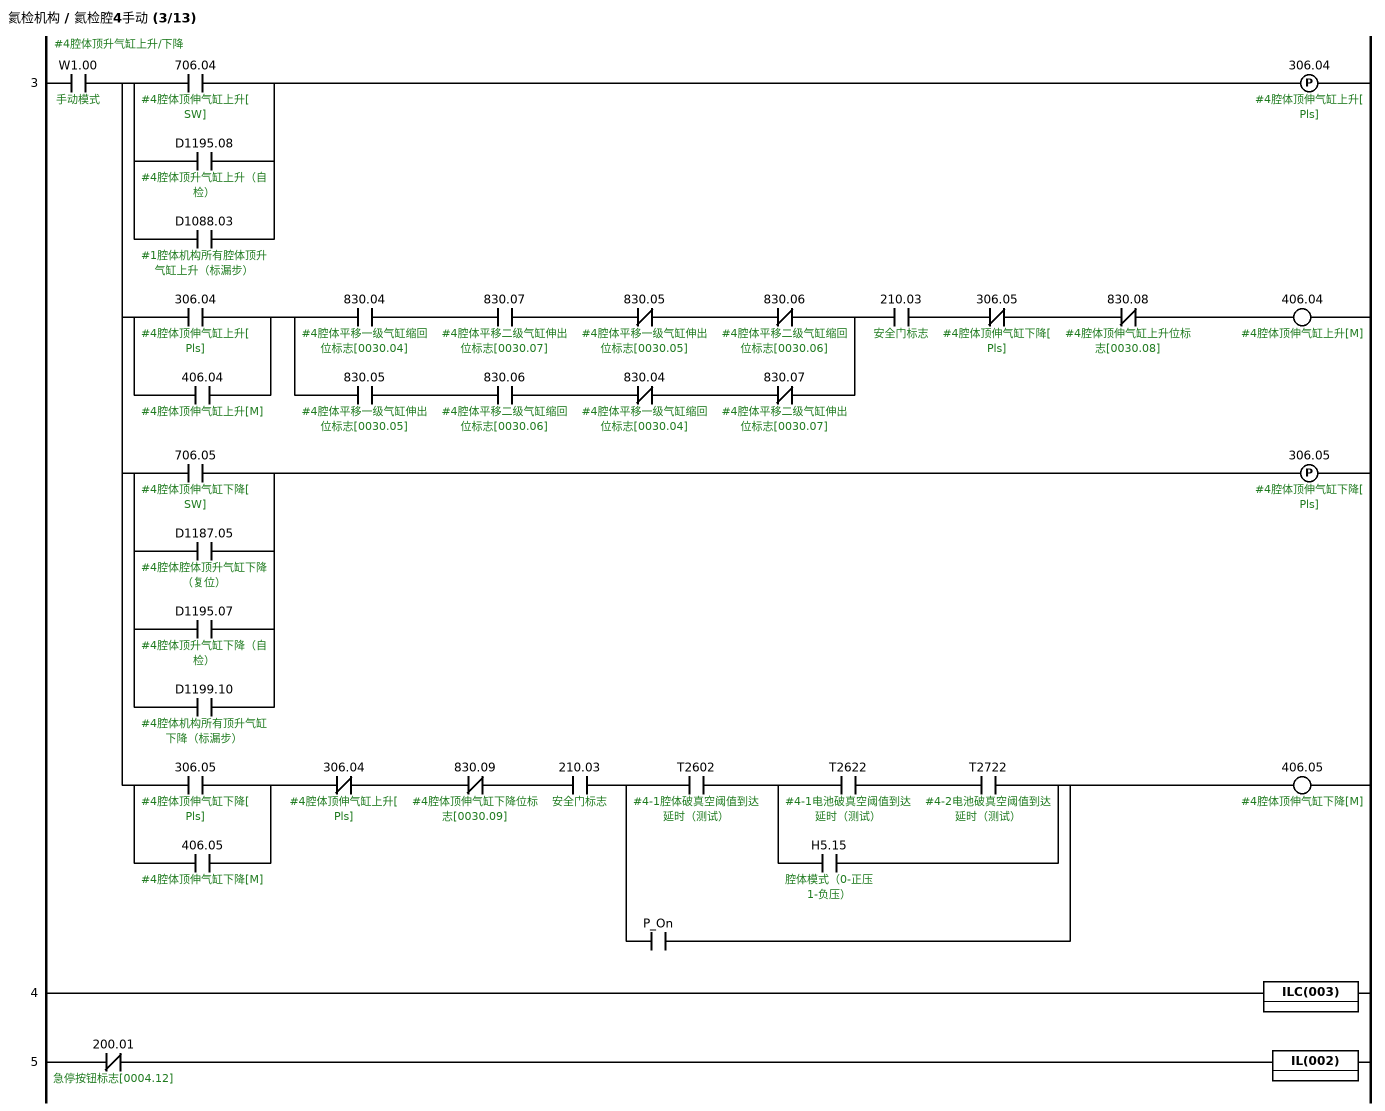
; rung 3: #4腔体顶升气缸上升/下降
LD W1.00  ; 手动模式
OUT TR0
LD 706.04  ; #4腔体顶伸气缸上升[SW]
OR D1195.08  ; #4腔体顶升气缸上升（自检）
OR D1088.03  ; #1腔体机构所有腔体顶升气缸上升（标漏步）
ANDLD
DIFU(013) 306.04  ; #4腔体顶伸气缸上升[Pls]
LD TR0
LD 306.04  ; #4腔体顶伸气缸上升[Pls]
OR 406.04  ; #4腔体顶伸气缸上升[M]
ANDLD
LD 830.04  ; #4腔体平移一级气缸缩回位标志[0030.04]
AND 830.07  ; #4腔体平移二级气缸伸出位标志[0030.07]
ANDNOT 830.05  ; #4腔体平移一级气缸伸出位标志[0030.05]
ANDNOT 830.06  ; #4腔体平移二级气缸缩回位标志[0030.06]
LD 830.05  ; #4腔体平移一级气缸伸出位标志[0030.05]
AND 830.06  ; #4腔体平移二级气缸缩回位标志[0030.06]
ANDNOT 830.04  ; #4腔体平移一级气缸缩回位标志[0030.04]
ANDNOT 830.07  ; #4腔体平移二级气缸伸出位标志[0030.07]
ORLD
ANDLD
AND 210.03  ; 安全门标志
ANDNOT 306.05  ; #4腔体顶伸气缸下降[Pls]
ANDNOT 830.08  ; #4腔体顶伸气缸上升位标志[0030.08]
OUT 406.04  ; #4腔体顶伸气缸上升[M]
LD TR0
LD 706.05  ; #4腔体顶伸气缸下降[SW]
OR D1187.05  ; #4腔体腔体顶升气缸下降（复位）
OR D1195.07  ; #4腔体顶升气缸下降（自检）
OR D1199.10  ; #4腔体机构所有顶升气缸下降（标漏步）
ANDLD
DIFU(013) 306.05  ; #4腔体顶伸气缸下降[Pls]
LD TR0
LD 306.05  ; #4腔体顶伸气缸下降[Pls]
OR 406.05  ; #4腔体顶伸气缸下降[M]
ANDLD
ANDNOT 306.04  ; #4腔体顶伸气缸上升[Pls]
ANDNOT 830.09  ; #4腔体顶伸气缸下降位标志[0030.09]
AND 210.03  ; 安全门标志
LD T2602  ; #4-1腔体破真空阈值到达延时（测试）
LD T2622  ; #4-1电池破真空阈值到达延时（测试）
AND T2722  ; #4-2电池破真空阈值到达延时（测试）
OR H5.15  ; 腔体模式（0-正压 1-负压）
ANDLD
OR P_On
ANDLD
OUT 406.05  ; #4腔体顶伸气缸下降[M]
; rung 4
ILC(003)
; rung 5
LDNOT 200.01  ; 急停按钮标志[0004.12]
IL(002)

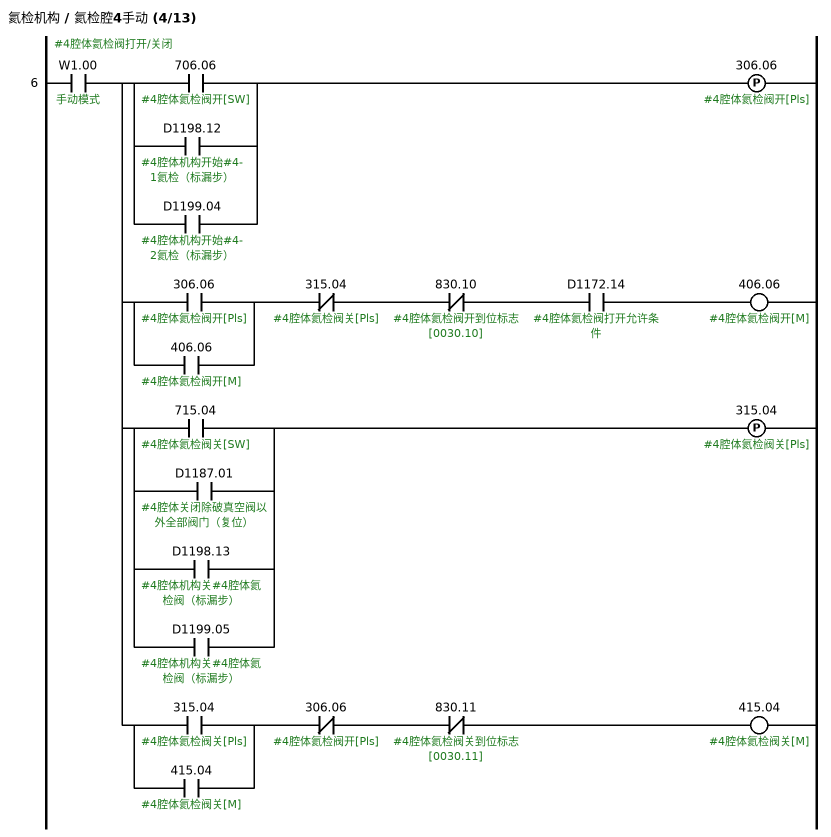
; rung 6: #4腔体氦检阀打开/关闭
LD W1.00  ; 手动模式
OUT TR0
LD 706.06  ; #4腔体氦检阀开[SW]
OR D1198.12  ; #4腔体机构开始#4-1氦检（标漏步）
OR D1199.04  ; #4腔体机构开始#4-2氦检（标漏步）
ANDLD
DIFU(013) 306.06  ; #4腔体氦检阀开[Pls]
LD TR0
LD 306.06  ; #4腔体氦检阀开[Pls]
OR 406.06  ; #4腔体氦检阀开[M]
ANDLD
ANDNOT 315.04  ; #4腔体氦检阀关[Pls]
ANDNOT 830.10  ; #4腔体氦检阀开到位标志[0030.10]
AND D1172.14  ; #4腔体氦检阀打开允许条件
OUT 406.06  ; #4腔体氦检阀开[M]
LD TR0
LD 715.04  ; #4腔体氦检阀关[SW]
OR D1187.01  ; #4腔体关闭除破真空阀以外全部阀门（复位）
OR D1198.13  ; #4腔体机构关#4腔体氦检阀（标漏步）
OR D1199.05  ; #4腔体机构关#4腔体氦检阀（标漏步）
ANDLD
DIFU(013) 315.04  ; #4腔体氦检阀关[Pls]
LD TR0
LD 315.04  ; #4腔体氦检阀关[Pls]
OR 415.04  ; #4腔体氦检阀关[M]
ANDLD
ANDNOT 306.06  ; #4腔体氦检阀开[Pls]
ANDNOT 830.11  ; #4腔体氦检阀关到位标志[0030.11]
OUT 415.04  ; #4腔体氦检阀关[M]

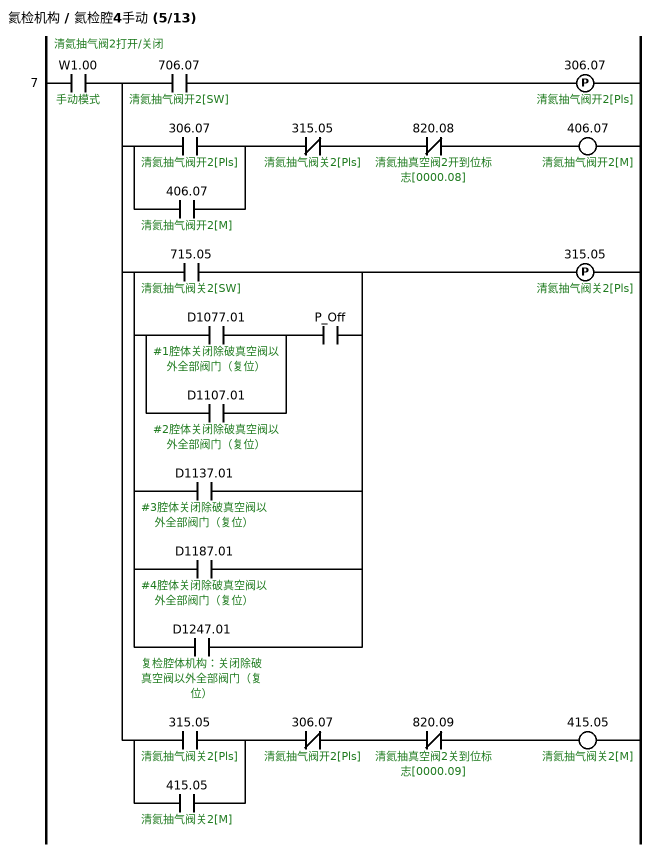
; rung 7: 清氦抽气阀2打开/关闭
LD W1.00  ; 手动模式
OUT TR0
AND 706.07  ; 清氦抽气阀开2[SW]
DIFU(013) 306.07  ; 清氦抽气阀开2[Pls]
LD TR0
LD 306.07  ; 清氦抽气阀开2[Pls]
OR 406.07  ; 清氦抽气阀开2[M]
ANDLD
ANDNOT 315.05  ; 清氦抽气阀关2[Pls]
ANDNOT 820.08  ; 清氦抽真空阀2开到位标志[0000.08]
OUT 406.07  ; 清氦抽气阀开2[M]
LD TR0
LD 715.05  ; 清氦抽气阀关2[SW]
LD D1077.01  ; #1腔体关闭除破真空阀以外全部阀门（复位）
OR D1107.01  ; #2腔体关闭除破真空阀以外全部阀门（复位）
AND P_Off
ORLD
OR D1137.01  ; #3腔体关闭除破真空阀以外全部阀门（复位）
OR D1187.01  ; #4腔体关闭除破真空阀以外全部阀门（复位）
OR D1247.01  ; 复检腔体机构：关闭除破真空阀以外全部阀门（复位）
ANDLD
DIFU(013) 315.05  ; 清氦抽气阀关2[Pls]
LD TR0
LD 315.05  ; 清氦抽气阀关2[Pls]
OR 415.05  ; 清氦抽气阀关2[M]
ANDLD
ANDNOT 306.07  ; 清氦抽气阀开2[Pls]
ANDNOT 820.09  ; 清氦抽真空阀2关到位标志[0000.09]
OUT 415.05  ; 清氦抽气阀关2[M]

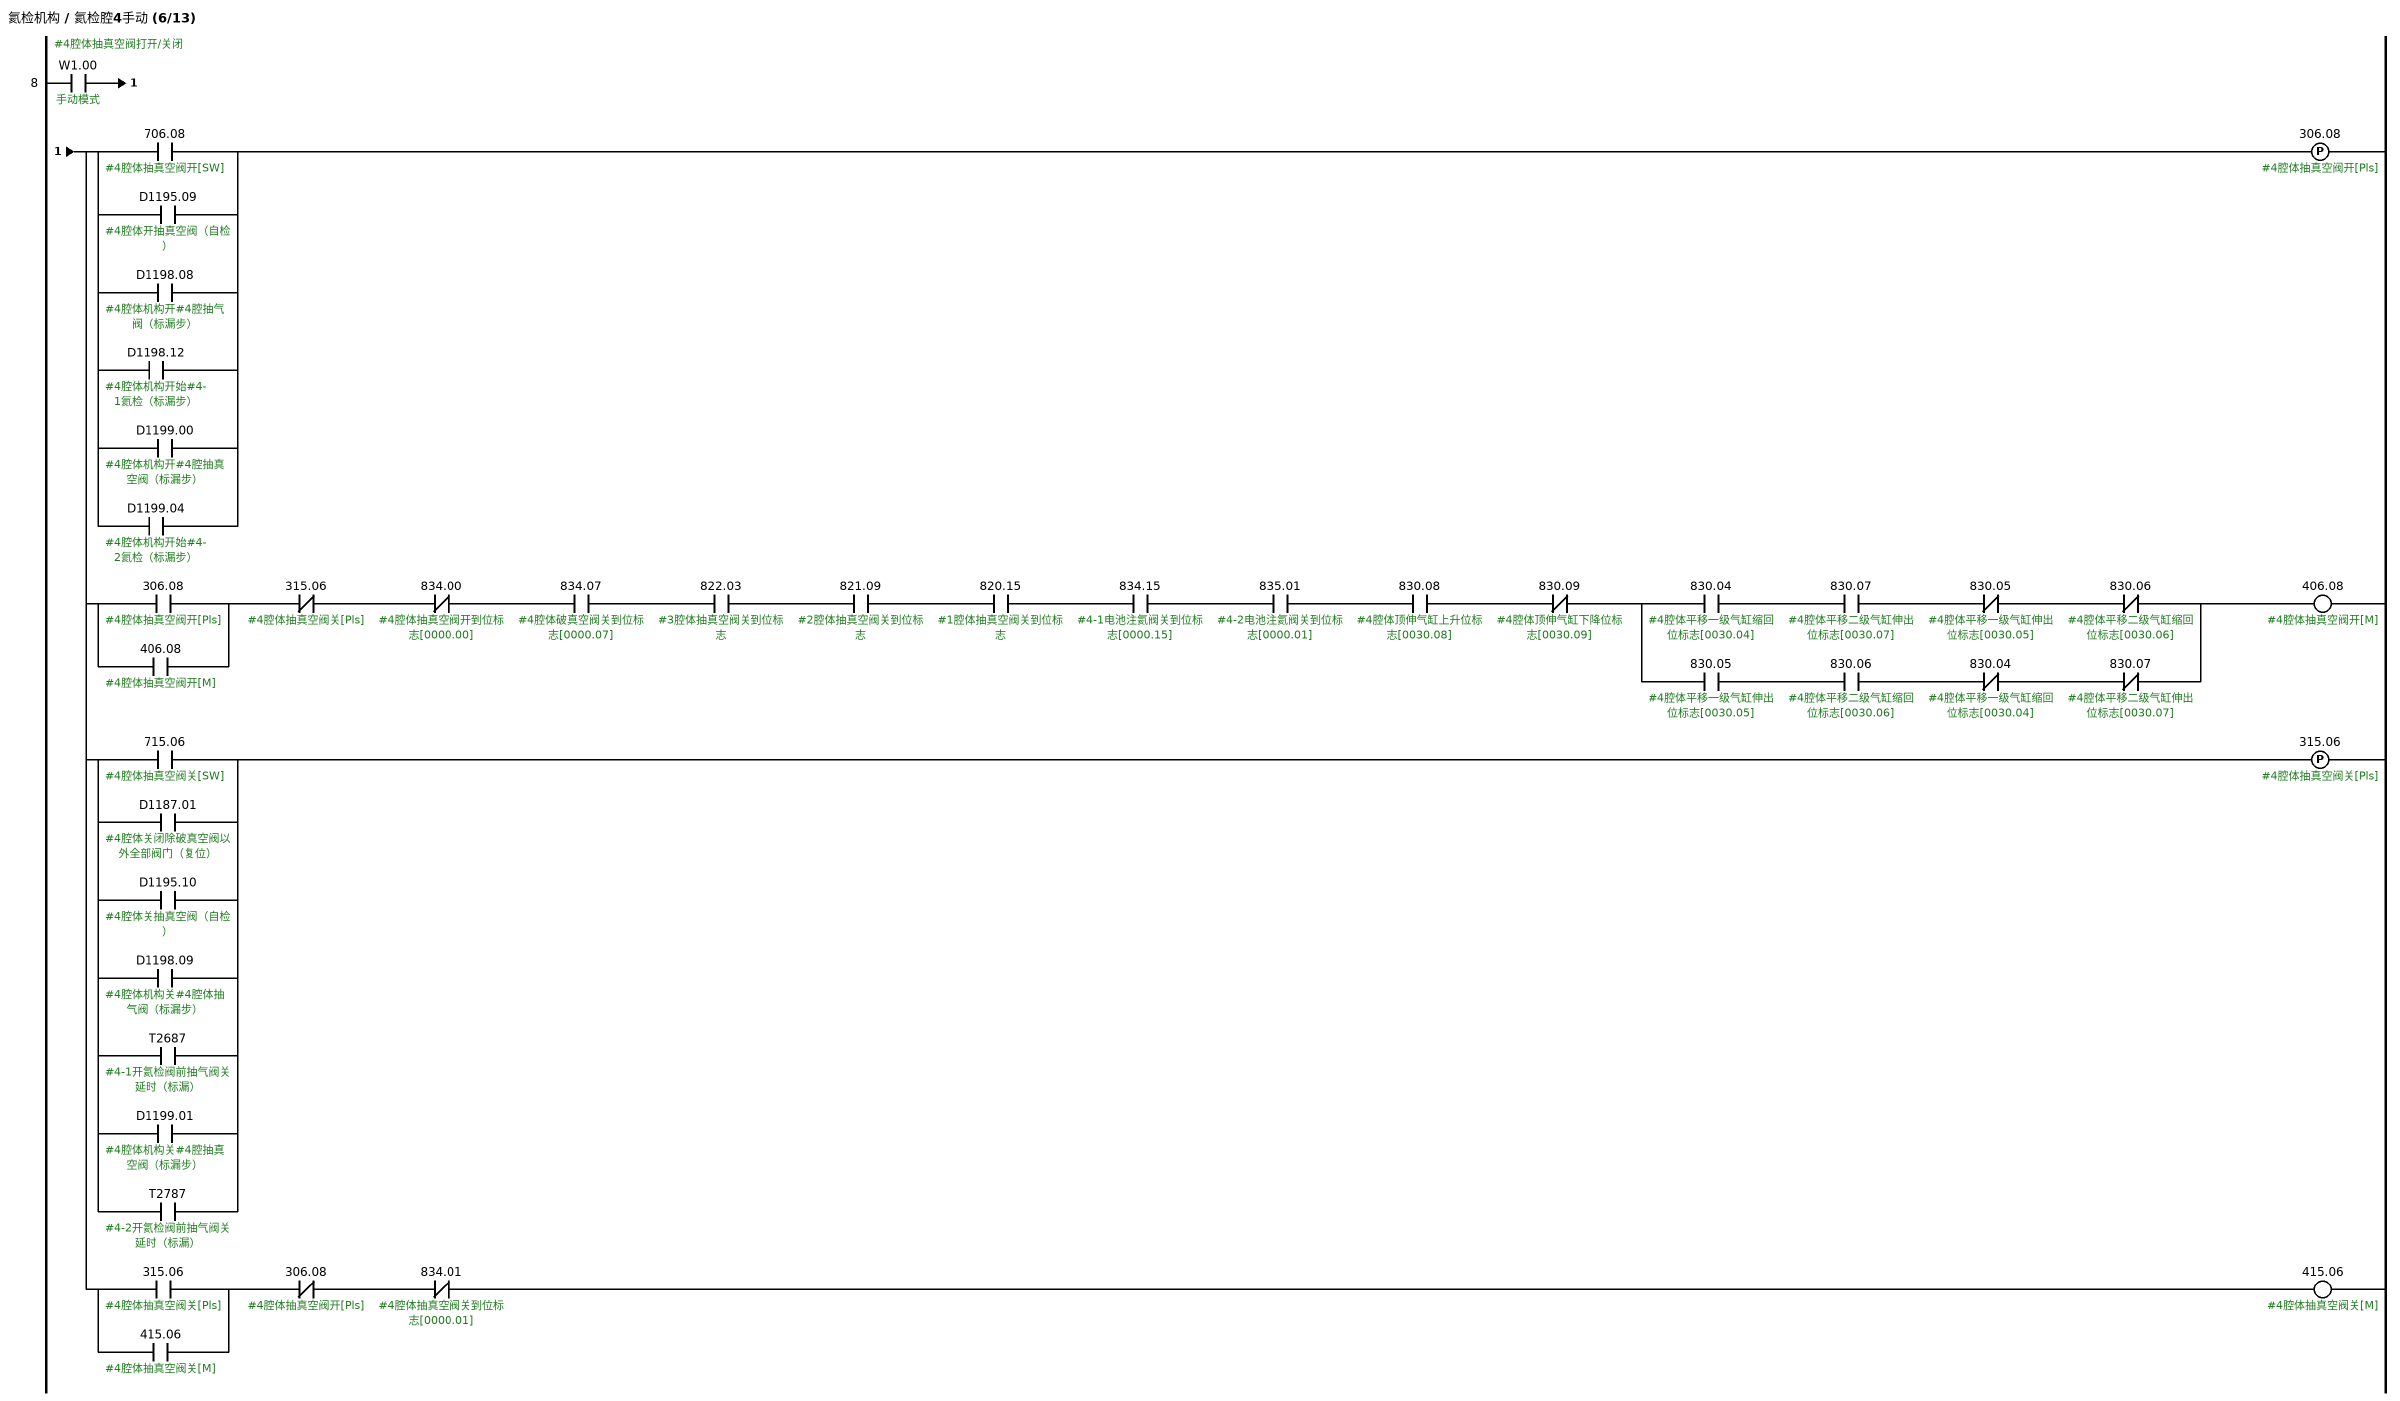
; rung 8: #4腔体抽真空阀打开/关闭
LD W1.00  ; 手动模式
OUT TR0
LD 706.08  ; #4腔体抽真空阀开[SW]
OR D1195.09  ; #4腔体开抽真空阀（自检）
OR D1198.08  ; #4腔体机构开#4腔抽气阀（标漏步）
OR D1198.12  ; #4腔体机构开始#4-1氦检（标漏步）
OR D1199.00  ; #4腔体机构开#4腔抽真空阀（标漏步）
OR D1199.04  ; #4腔体机构开始#4-2氦检（标漏步）
ANDLD
DIFU(013) 306.08  ; #4腔体抽真空阀开[Pls]
LD TR0
LD 306.08  ; #4腔体抽真空阀开[Pls]
OR 406.08  ; #4腔体抽真空阀开[M]
ANDLD
ANDNOT 315.06  ; #4腔体抽真空阀关[Pls]
ANDNOT 834.00  ; #4腔体抽真空阀开到位标志[0000.00]
AND 834.07  ; #4腔体破真空阀关到位标志[0000.07]
AND 822.03  ; #3腔体抽真空阀关到位标志
AND 821.09  ; #2腔体抽真空阀关到位标志
AND 820.15  ; #1腔体抽真空阀关到位标志
AND 834.15  ; #4-1电池注氦阀关到位标志[0000.15]
AND 835.01  ; #4-2电池注氦阀关到位标志[0000.01]
AND 830.08  ; #4腔体顶伸气缸上升位标志[0030.08]
ANDNOT 830.09  ; #4腔体顶伸气缸下降位标志[0030.09]
LD 830.04  ; #4腔体平移一级气缸缩回位标志[0030.04]
AND 830.07  ; #4腔体平移二级气缸伸出位标志[0030.07]
ANDNOT 830.05  ; #4腔体平移一级气缸伸出位标志[0030.05]
ANDNOT 830.06  ; #4腔体平移二级气缸缩回位标志[0030.06]
LD 830.05  ; #4腔体平移一级气缸伸出位标志[0030.05]
AND 830.06  ; #4腔体平移二级气缸缩回位标志[0030.06]
ANDNOT 830.04  ; #4腔体平移一级气缸缩回位标志[0030.04]
ANDNOT 830.07  ; #4腔体平移二级气缸伸出位标志[0030.07]
ORLD
ANDLD
OUT 406.08  ; #4腔体抽真空阀开[M]
LD TR0
LD 715.06  ; #4腔体抽真空阀关[SW]
OR D1187.01  ; #4腔体关闭除破真空阀以外全部阀门（复位）
OR D1195.10  ; #4腔体关抽真空阀（自检）
OR D1198.09  ; #4腔体机构关#4腔体抽气阀（标漏步）
OR T2687  ; #4-1开氦检阀前抽气阀关延时（标漏）
OR D1199.01  ; #4腔体机构关#4腔抽真空阀（标漏步）
OR T2787  ; #4-2开氦检阀前抽气阀关延时（标漏）
ANDLD
DIFU(013) 315.06  ; #4腔体抽真空阀关[Pls]
LD TR0
LD 315.06  ; #4腔体抽真空阀关[Pls]
OR 415.06  ; #4腔体抽真空阀关[M]
ANDLD
ANDNOT 306.08  ; #4腔体抽真空阀开[Pls]
ANDNOT 834.01  ; #4腔体抽真空阀关到位标志[0000.01]
OUT 415.06  ; #4腔体抽真空阀关[M]

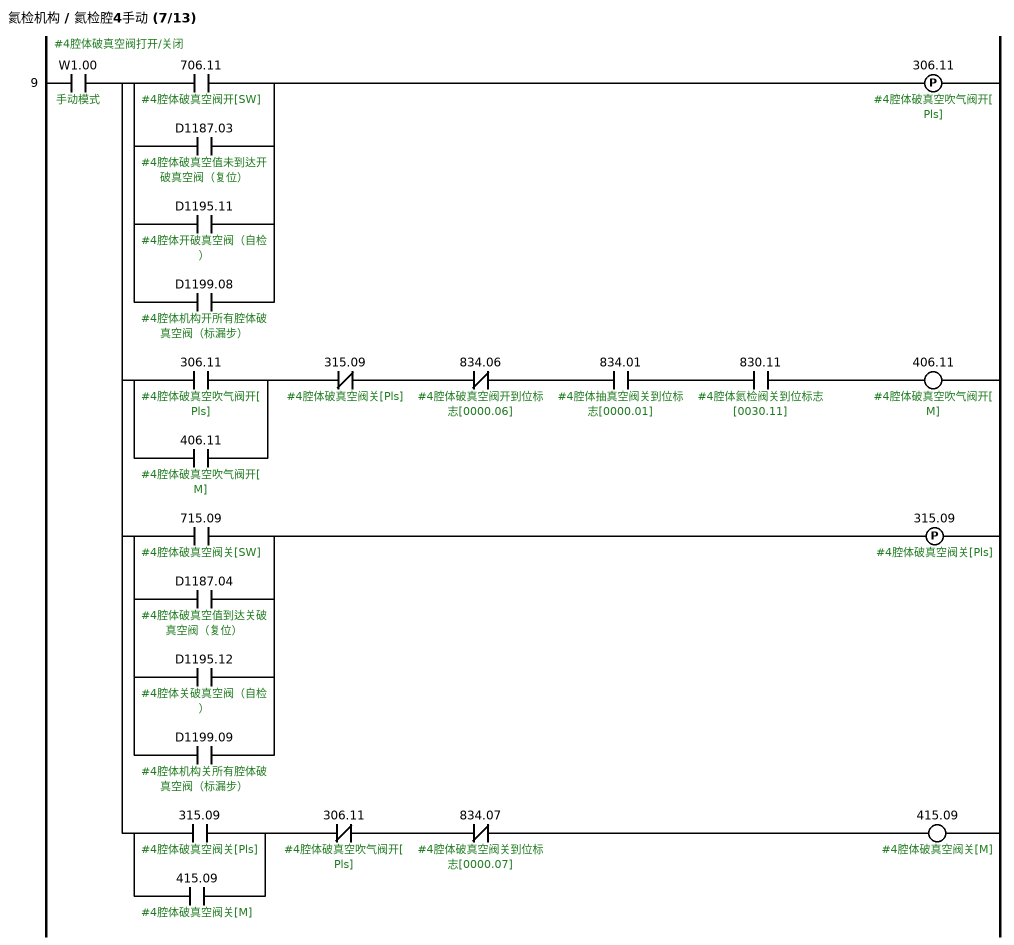
; rung 9: #4腔体破真空阀打开/关闭
LD W1.00  ; 手动模式
OUT TR0
LD 706.11  ; #4腔体破真空阀开[SW]
OR D1187.03  ; #4腔体破真空值未到达开破真空阀（复位）
OR D1195.11  ; #4腔体开破真空阀（自检）
OR D1199.08  ; #4腔体机构开所有腔体破真空阀（标漏步）
ANDLD
DIFU(013) 306.11  ; #4腔体破真空吹气阀开[Pls]
LD TR0
LD 306.11  ; #4腔体破真空吹气阀开[Pls]
OR 406.11  ; #4腔体破真空吹气阀开[M]
ANDLD
ANDNOT 315.09  ; #4腔体破真空阀关[Pls]
ANDNOT 834.06  ; #4腔体破真空阀开到位标志[0000.06]
AND 834.01  ; #4腔体抽真空阀关到位标志[0000.01]
AND 830.11  ; #4腔体氦检阀关到位标志[0030.11]
OUT 406.11  ; #4腔体破真空吹气阀开[M]
LD TR0
LD 715.09  ; #4腔体破真空阀关[SW]
OR D1187.04  ; #4腔体破真空值到达关破真空阀（复位）
OR D1195.12  ; #4腔体关破真空阀（自检）
OR D1199.09  ; #4腔体机构关所有腔体破真空阀（标漏步）
ANDLD
DIFU(013) 315.09  ; #4腔体破真空阀关[Pls]
LD TR0
LD 315.09  ; #4腔体破真空阀关[Pls]
OR 415.09  ; #4腔体破真空阀关[M]
ANDLD
ANDNOT 306.11  ; #4腔体破真空吹气阀开[Pls]
ANDNOT 834.07  ; #4腔体破真空阀关到位标志[0000.07]
OUT 415.09  ; #4腔体破真空阀关[M]

